		(* UPS Überwachung *)
		UPS.st_config.b_config_fertig := FALSE;
		UPS.st_config.b_station_aktiv := TRUE;
		UPS.st_config.i16_meld_startindex := 440;		(*-445*)
		UPS.st_config.str_beschreibung := ' ';
		UPS.st_config.str_instanz_name := 'UPS Überwachung';
		UPS.st_config.b_config_fertig := TRUE;

		(*Einpresskraftkontroller *)
		einpresskraft_kontroller.st_config.b_config_fertig := FALSE;
		einpresskraft_kontroller.st_config.b_station_aktiv := TRUE;
		einpresskraft_kontroller.st_config.i16_meld_startindex := 460;
		einpresskraft_kontroller.st_config.str_beschreibung := ' ';
		einpresskraft_kontroller.st_config.str_instanz_name := 'Einpresskraftkontroller';

		CASE gst_datensatz.st_md.i16_typ_zelle OF
			KEINE_ZELLE:
				gst_datensatz.st_band.st_einpressen.st_einstellungen.enu_modus := KEIN_MODUS;
			BESTUECKZELLE_1700:
				gst_datensatz.st_band.st_einpressen.st_einstellungen.enu_modus := F_MAXWERT;
			BESTUECKZELLE_1720:
				gst_datensatz.st_band.st_einpressen.st_einstellungen.enu_modus := F_MAXWERT;
			RASTERFOLIE:
				gst_datensatz.st_band.st_einpressen.st_einstellungen.enu_modus := KEIN_MODUS;
		END_CASE

		einpresskraft_kontroller.st_config.b_config_fertig := TRUE;
		
		(* Kraftmessdose Kanal 1*)
		kraftmessdose.fb.st_config.b_config_fertig := FALSE;
		kraftmessdose.fb.st_config.b_station_aktiv := TRUE;
		kraftmessdose.fb.st_config.i16_meld_startindex := 480;
		kraftmessdose.fb.st_config.str_beschreibung := ' ';
		kraftmessdose.fb.st_config.str_instanz_name := 'Kraftmessdose Kanal 1';
		kraftmessdose.fb.st_config.b_config_fertig := TRUE;
		
		(* Nockenschaltwerk Bestückachse *)
		nockenschaltwerk_bestueckachse.st_config.b_config_fertig := FALSE;
		nockenschaltwerk_bestueckachse.st_config.b_station_aktiv := TRUE;
		nockenschaltwerk_bestueckachse.st_config.i16_meld_startindex := 500;
		nockenschaltwerk_bestueckachse.st_config.str_beschreibung := ' ';
		nockenschaltwerk_bestueckachse.st_config.str_instanz_name := 'Nockenschaltwerk Bestückachse';
		nockenschaltwerk_bestueckachse.st_config.b_config_fertig := TRUE;
		
		(* Nockenschaltwerk Z-Achse *)
		(* 520 *)
		
		(* Nockenschaltwerk Y-Achse *)
		(* 540 *)
		
		(* Frei *)
		(* 560 *)

		(* Safety *)
		safety.st_config.b_config_fertig := FALSE;
		safety.st_config.b_station_aktiv := TRUE;
		safety.st_config.i16_meld_startindex := 580;
		safety.st_config.str_beschreibung := ' ';
		safety.st_config.str_instanz_name := 'Safety';
		safety.st_config.b_config_fertig := TRUE;
		
		(* XML-Server *)
		xml_server.st_config.b_config_fertig := FALSE;
		xml_server.st_config.b_station_aktiv := TRUE;
		xml_server.st_config.i16_meld_startindex := 620;
		xml_server.st_config.str_beschreibung := ' ';
		xml_server.st_config.str_instanz_name := 'XML-Server';
		xml_server.st_config.b_config_fertig := TRUE;

		(* Kurvenscheibeneditor *)
		fb_edit_mfps_bestuecken_z.st_config.b_config_fertig := FALSE;
		fb_edit_mfps_bestuecken_z.st_config.b_station_aktiv := TRUE;
		fb_edit_mfps_bestuecken_z.st_config.i16_meld_startindex := 640;
		fb_edit_mfps_bestuecken_z.st_config.str_beschreibung := ' ';
		fb_edit_mfps_bestuecken_z.st_config.str_instanz_name := 'Kurvenscheibeneditor Bestücken Z-Achse';
		fb_edit_mfps_bestuecken_z.st_config.b_config_fertig := TRUE;
		
		fb_edit_mfps_bestuecken_y.st_config.b_config_fertig := FALSE;
		fb_edit_mfps_bestuecken_y.st_config.b_station_aktiv := TRUE;
		fb_edit_mfps_bestuecken_y.st_config.i16_meld_startindex := 660;
		fb_edit_mfps_bestuecken_y.st_config.str_beschreibung := ' ';
		fb_edit_mfps_bestuecken_y.st_config.str_instanz_name := 'Kurvenscheibeneditor Bestücken Y-Achse';
		fb_edit_mfps_bestuecken_y.st_config.b_config_fertig := TRUE;
		
		fb_edit_mfps_yz_tisch.st_config.b_config_fertig := FALSE;
		fb_edit_mfps_yz_tisch.st_config.b_station_aktiv := TRUE;
		fb_edit_mfps_yz_tisch.st_config.i16_meld_startindex := 680;
		fb_edit_mfps_yz_tisch.st_config.str_beschreibung := ' ';
		fb_edit_mfps_yz_tisch.st_config.str_instanz_name := 'Kurvenscheibeneditor YZ-Tisch';
		fb_edit_mfps_yz_tisch.st_config.b_config_fertig := TRUE;

		fb_edit_mfps_bestuecken_b.st_config.b_config_fertig := FALSE;
		fb_edit_mfps_bestuecken_b.st_config.b_station_aktiv := TRUE;
		fb_edit_mfps_bestuecken_b.st_config.i16_meld_startindex := 860;
		fb_edit_mfps_bestuecken_b.st_config.str_beschreibung := ' ';
		fb_edit_mfps_bestuecken_b.st_config.str_instanz_name := 'Kurvenscheibeneditor Bestücken B-Achse';
		fb_edit_mfps_bestuecken_b.st_config.b_config_fertig := TRUE;

		fb_camtable_bestueckachse.st_config.b_config_fertig := FALSE;
		fb_camtable_bestueckachse.st_config.b_station_aktiv := TRUE;
		fb_camtable_bestueckachse.st_config.i16_meld_startindex := 880;
		fb_camtable_bestueckachse.st_config.str_beschreibung := ' ';
		fb_camtable_bestueckachse.st_config.str_instanz_name := 'Kurvenscheibeneditor Bestückachse';
		fb_camtable_bestueckachse.st_config.b_config_fertig := TRUE;

		(* Bestückbildgenerierung *)
		bbgen.st_config.b_config_fertig := FALSE;
		bbgen.st_config.b_station_aktiv := TRUE;
		bbgen.st_config.i16_meld_startindex := 700;
		bbgen.st_config.str_beschreibung := ' ';
		bbgen.st_config.str_instanz_name := 'Bestückbildgenerierung';
		bbgen.st_config.b_config_fertig := TRUE;
		
		(* Barcodereader *)
		barcode.fb.st_config.b_config_fertig := FALSE;
		barcode.fb.st_config.b_station_aktiv := TRUE;
		barcode.fb.st_config.i16_meld_startindex := 720;
		barcode.fb.st_config.str_beschreibung := ' ';
		barcode.fb.st_config.str_instanz_name := 'Barcodereader';
		barcode.fb.st_config.b_config_fertig := TRUE;
		
		(* Ballufftagreader *)
		balluff_tag_reader.fb.st_config.b_config_fertig := FALSE;
		balluff_tag_reader.fb.st_config.b_station_aktiv := TRUE;
		balluff_tag_reader.fb.st_config.i16_meld_startindex := 740;
		balluff_tag_reader.fb.st_config.str_beschreibung := ' ';
		balluff_tag_reader.fb.st_config.str_instanz_name := 'Ballufftagreader';
		balluff_tag_reader.fb.st_config.b_config_fertig := TRUE;

		(* WT-Transport Warteposition 1720 *)
		wt_transport_warteposition_1720.st_config.b_config_fertig := FALSE;
		wt_transport_warteposition_1720.st_config.i16_meld_startindex := 760;
		wt_transport_warteposition_1720.st_config.str_beschreibung := ' ';
		wt_transport_warteposition_1720.st_config.str_instanz_name := 'WT-Transport Warteposition 1720';
		wt_transport_warteposition_1720.st_config.b_config_fertig := TRUE;
		
		(* WT-Transport Beladestation 1720 *)
		wt_transport_beladen_1720.st_config.b_config_fertig := FALSE;
		wt_transport_beladen_1720.st_config.i16_meld_startindex := 780;
		wt_transport_beladen_1720.st_config.str_beschreibung := ' ';
		wt_transport_beladen_1720.st_config.str_instanz_name := 'WT-Transport Beladestation 1720';
		wt_transport_beladen_1720.st_config.b_config_fertig := TRUE;
		
		(* Rasterfolienmontge *)
		rasterfolienmontage.st_config.b_config_fertig := FALSE;
		rasterfolienmontage.st_config.b_station_aktiv := TRUE;
		rasterfolienmontage.st_config.i16_meld_startindex := 800;
		rasterfolienmontage.st_config.str_beschreibung := ' ';
		rasterfolienmontage.st_config.str_instanz_name := 'Rasterfolienmontge';
		rasterfolienmontage.st_config.b_config_fertig := TRUE;
		
		(* Rasterfolieneinzug *)
		rasterfolieneinzug.st_config.b_config_fertig := FALSE;
		rasterfolieneinzug.st_config.b_station_aktiv := TRUE;
		rasterfolieneinzug.st_config.i16_meld_startindex := 820;
		rasterfolieneinzug.st_config.str_beschreibung := ' ';
		rasterfolieneinzug.st_config.str_instanz_name := 'Rasterfolieneinzug';
		rasterfolieneinzug.st_config.b_config_fertig := TRUE;

		(*Tag lesen und schreiben *)
		Lesen_Schreiben_Tag.st_config.b_config_fertig := FALSE;
		Lesen_Schreiben_Tag.st_config.b_station_aktiv := TRUE;
		Lesen_Schreiben_Tag.st_config.i16_meld_startindex := 840;
		Lesen_Schreiben_Tag.st_config.str_beschreibung := ' ';
		Lesen_Schreiben_Tag.st_config.str_instanz_name := 'Tag lesen und schreiben';
		Lesen_Schreiben_Tag.st_config.b_config_fertig := TRUE;

		(* Wartung *)
		wartung.st_config.b_config_fertig := FALSE;
		wartung.st_config.b_station_aktiv := TRUE;
		wartung.st_config.i16_meld_startindex := 920;
		wartung.st_config.str_beschreibung := ' ';
		wartung.st_config.str_instanz_name := 'Wartung';
		wartung.st_config.b_config_fertig := TRUE;

		(*Service *)
		Service.st_config.b_config_fertig := FALSE;
		Service.st_config.b_station_aktiv := TRUE;
		Service.st_config.i16_meld_startindex := 900;
		Service.st_config.str_beschreibung := ' ';
		Service.st_config.str_instanz_name := 'Service';
		Service.st_config.b_config_fertig := TRUE;

		(*TouchProbe *)
		ST_TouchProbe.st_config.b_config_fertig := FALSE;
		ST_TouchProbe.st_config.b_station_aktiv := TRUE;
		ST_TouchProbe.st_config.i16_meld_startindex := 940;
		ST_TouchProbe.st_config.str_beschreibung := ' ';
		ST_TouchProbe.st_config.str_instanz_name := 'TouchProbe';
		ST_TouchProbe.st_config.b_config_fertig := TRUE;

		(*AutocheckinDaten *)
		ST_AutoCheckIn.fb_AutocheckinDaten.st_config.b_config_fertig:= FALSE;
		ST_AutoCheckIn.fb_AutocheckinDaten.st_config.b_station_aktiv:= TRUE;
		ST_AutoCheckIn.fb_AutocheckinDaten.st_config.i16_meld_startindex:=	960;
		ST_AutoCheckIn.fb_AutocheckinDaten.st_config.str_beschreibung:= ' ';
		ST_AutoCheckIn.fb_AutocheckinDaten.st_config.str_instanz_name:=	'AutoCheckInDaten';
		ST_AutoCheckIn.fb_AutocheckinDaten.st_config.b_config_fertig:= TRUE;

		(* WT-Transport Warteposition Achse 1700 *)
		wt_transport_warteposition_1700.st_config.b_config_fertig := FALSE;
		wt_transport_warteposition_1700.st_config.i16_meld_startindex := 400;
		wt_transport_warteposition_1700.st_config.str_beschreibung := ' ';
		wt_transport_warteposition_1700.st_config.str_instanz_name := 'WT-Transport Warteposition 1700';
		wt_transport_warteposition_1700.st_config.b_config_fertig := TRUE;
		
		(* WT-Transport Beladestation Achse 1700 *)
		wt_transport_beladen_achse_1700.st_config.b_config_fertig := FALSE;
		wt_transport_beladen_achse_1700.st_config.i16_meld_startindex := 420;
		wt_transport_beladen_achse_1700.st_config.str_beschreibung := ' ';
		wt_transport_beladen_achse_1700.st_config.str_instanz_name := 'WT-Transport Beladestation Achse 1700';
		wt_transport_beladen_achse_1700.st_config.b_config_fertig := TRUE;

		(* EtherCAT Diagnose *)
		Index:=1;
		EtherCatDiag[Index].st_config.b_config_fertig := FALSE;
		EtherCatDiag[Index].st_config.b_station_aktiv := TRUE;
		EtherCatDiag[Index].st_config.i16_meld_startindex := 980;
		EtherCatDiag[Index].st_config.str_beschreibung := ' ';
		EtherCatDiag[Index].st_config.str_instanz_name := 'Grundmaschine';
		EtherCatDiag[Index].st_config.b_config_fertig := TRUE;

		(* EtherCAT Diagnose *)
		Index:=2;
		EtherCatDiag[Index].st_config.b_config_fertig := FALSE;
		EtherCatDiag[Index].st_config.b_station_aktiv := TRUE;
		EtherCatDiag[Index].st_config.i16_meld_startindex := 985;
		EtherCatDiag[Index].st_config.str_beschreibung := ' ';
		EtherCatDiag[Index].st_config.str_instanz_name := 'Hublift links';
		EtherCatDiag[Index].st_config.b_config_fertig := TRUE;

		(* EtherCAT Diagnose *)
		Index:=3;
		EtherCatDiag[Index].st_config.b_config_fertig := FALSE;
		EtherCatDiag[Index].st_config.b_station_aktiv := TRUE;
		EtherCatDiag[Index].st_config.i16_meld_startindex := 990;
		EtherCatDiag[Index].st_config.str_beschreibung := ' ';
		EtherCatDiag[Index].st_config.str_instanz_name := 'Hublift rechts';
		EtherCatDiag[Index].st_config.b_config_fertig := TRUE;

		(* EtherCAT Diagnose *)
		Index:=4;
		EtherCatDiag[Index].st_config.b_config_fertig := FALSE;
		EtherCatDiag[Index].st_config.b_station_aktiv := TRUE;
		EtherCatDiag[Index].st_config.i16_meld_startindex := 995;
		EtherCatDiag[Index].st_config.str_beschreibung := ' ';
		EtherCatDiag[Index].st_config.str_instanz_name := 'Bandeinzug';
		EtherCatDiag[Index].st_config.b_config_fertig := TRUE;

		(* Melde-Arrays rücksetzen *)
		FOR i := 0 TO SIZEOF (garr_stoermeldungen) / SIZEOF (garr_stoermeldungen[0]) - 1 BY 1 DO
			garr_stoermeldungen[i] := 0;
		END_FOR
		FOR i := 0 TO SIZEOF (garr_betriebsmeldungen) / SIZEOF (garr_betriebsmeldungen[0]) - 1 BY 1 DO
			garr_betriebsmeldungen[i] := 0;
		END_FOR
ELSE
	b_config_fertig := TRUE;
END_IF

		
		
END_PROGRAM

(* POU Gemeinsamkeiten17xx/Initialisierung/Startup/ST_Datainit_Zylinder, ST *)
PROGRAM ST_Datainit_Zylinder
VAR
	b_config_fertig			: BOOL := FALSE;
END_VAR
IF	NOT zyl_wt_zentrierer_tisch.fb.st_config.b_config_fertig OR
	NOT zyl_wt_stopper_tisch.fb.st_config.b_config_fertig OR
	NOT zyl_wt_stopper_auslauf.fb.st_config.b_config_fertig OR
	NOT zyl_hublift_rechts_lift.fb.st_config.b_config_fertig OR
	NOT zyl_hublift_rechts_wt_einzug.fb.st_config.b_config_fertig OR
	NOT zyl_hublift_rechts_wt_klinke.fb.st_config.b_config_fertig OR
	NOT zyl_hublift_links_lift.fb.st_config.b_config_fertig OR
	NOT zyl_hublift_links_wt_einzug.fb.st_config.b_config_fertig OR
	NOT zyl_hublift_links_wt_klinke.fb.st_config.b_config_fertig OR
	NOT zyl_hublift_links_stopper.fb.st_config.b_config_fertig OR
	NOT zyl_hublift_links_eingriffschutz.fb.st_config.b_config_fertig OR
	NOT zyl_haspel_li_heben.fb.st_config.b_config_fertig OR
	NOT zyl_haspel_li_abspulen.fb.st_config.b_config_fertig OR
	NOT zyl_haspel_li_sperren.fb.st_config.b_config_fertig OR
	NOT zyl_haspel_re_heben.fb.st_config.b_config_fertig OR
	NOT zyl_haspel_re_abspulen.fb.st_config.b_config_fertig OR
	NOT zyl_haspel_re_sperren.fb.st_config.b_config_fertig OR
	NOT zyl_haspel_verschieben.fb.st_config.b_config_fertig OR
	NOT zyl_bandeinzuege_verschieben.fb.st_config.b_config_fertig OR
	NOT zyl_bawe_vorschub.fb.st_config.b_config_fertig OR
	NOT zyl_bawe_querschub.fb.st_config.b_config_fertig OR
	NOT zyl_bawe_faenger_li.fb.st_config.b_config_fertig OR
	NOT zyl_bawe_faenger_re.fb.st_config.b_config_fertig OR
	NOT zyl_bawe_halter_li.fb.st_config.b_config_fertig OR
	NOT zyl_bawe_halter_re.fb.st_config.b_config_fertig OR
	NOT zyl_wt_stopper_einlauf.fb.st_config.b_config_fertig OR
	NOT zyl_rafo_faenger.fb.st_config.b_config_fertig OR
	NOT zyl_rafo_klemmen.fb.st_config.b_config_fertig OR
	NOT zyl_rafo_vorschub.fb.st_config.b_config_fertig OR
	NOT zyl_rafo_kamm.fb.st_config.b_config_fertig OR
	NOT zyl_rafo_vorzentrierer.fb.st_config.b_config_fertig OR
	NOT zyl_Indexier_Bestueckpos.fb.st_config.b_config_fertig OR
	NOT zyl_Indexier_Einlauf.fb.st_config.b_config_fertig
	THEN

		(* WT Zentrierzylinder am Tisch *)
		zyl_wt_zentrierer_tisch.fb.st_config.b_config_fertig := FALSE;
		zyl_wt_zentrierer_tisch.fb.st_config.b_endlage1_aktiv := FALSE;
		zyl_wt_zentrierer_tisch.fb.st_config.b_endlage2_aktiv := FALSE;
		zyl_wt_zentrierer_tisch.fb.st_config.b_sensor1_aktiv := TRUE;
		zyl_wt_zentrierer_tisch.fb.st_config.b_sensor2_aktiv := TRUE;
		zyl_wt_zentrierer_tisch.fb.st_config.i16_gruppe := 3;
		zyl_wt_zentrierer_tisch.fb.st_config.i16_identnummer := 15;
		zyl_wt_zentrierer_tisch.fb.st_config.i16_meld_startindex := 2280;
		zyl_wt_zentrierer_tisch.fb.st_config.str_beschreibung := ' ';
		zyl_wt_zentrierer_tisch.fb.st_config.str_instanz_name := 'WT Zentrierzylinder am Tisch';
		zyl_wt_zentrierer_tisch.fb.st_config.str_zylinder_typ := '2V4E_EIN_AUS';
		zyl_wt_zentrierer_tisch.fb.st_config.t_ein_aus_fahrzeit := t#0ms;
		zyl_wt_zentrierer_tisch.fb.st_config.t_ueberwachungszeit := t#1000ms;
		zyl_wt_zentrierer_tisch.fb.st_config.i16_tzk_faktor_ausfahren := 100;
		zyl_wt_zentrierer_tisch.fb.st_config.i16_tzk_faktor_einfahren := 100;
		zyl_wt_zentrierer_tisch.fb.st_config.b_config_fertig := TRUE;
		
		(* WT Stoppzylinder am Tisch *)
		zyl_wt_stopper_tisch.fb.st_config.b_config_fertig := FALSE;
		zyl_wt_stopper_tisch.fb.st_config.b_endlage1_aktiv := FALSE;
		zyl_wt_stopper_tisch.fb.st_config.b_endlage2_aktiv := FALSE;
		zyl_wt_stopper_tisch.fb.st_config.b_sensor1_aktiv := TRUE;
		zyl_wt_stopper_tisch.fb.st_config.b_sensor2_aktiv := FALSE;
		zyl_wt_stopper_tisch.fb.st_config.i16_gruppe := 3;
		zyl_wt_stopper_tisch.fb.st_config.i16_identnummer := 16;
		zyl_wt_stopper_tisch.fb.st_config.i16_meld_startindex := 2300;
		zyl_wt_stopper_tisch.fb.st_config.str_beschreibung := ' ';
		zyl_wt_stopper_tisch.fb.st_config.str_instanz_name := 'WT Stoppzylinder am Tisch';

		zyl_wt_stopper_tisch.fb.st_config.t_ein_aus_fahrzeit := t#0ms;
		zyl_wt_stopper_tisch.fb.st_config.t_ueberwachungszeit := t#1000ms;
		zyl_wt_stopper_tisch.fb.st_config.i16_tzk_faktor_ausfahren := 100;
		zyl_wt_stopper_tisch.fb.st_config.i16_tzk_faktor_einfahren := 100;


		IF gst_Datensatz.st_md.b_anwahl_transport_achse THEN
			zyl_wt_stopper_tisch.fb.st_config.str_zylinder_typ := '1V0E_NO';
		ELSE
			zyl_wt_stopper_tisch.fb.st_config.str_zylinder_typ := '2V2E_EIN_AUS';
		END_IF

		zyl_wt_stopper_tisch.fb.st_config.b_config_fertig := TRUE;

		(* WT Stopperzylinder am Auslauf *)
		CASE gst_datensatz.st_md.i16_typ_zelle OF
			KEINE_ZELLE:
				;
			BESTUECKZELLE_1700, RASTERFOLIE:
				zyl_wt_stopper_auslauf.fb.st_config.b_config_fertig := FALSE;
				zyl_wt_stopper_auslauf.fb.st_config.b_endlage1_aktiv := FALSE;
				zyl_wt_stopper_auslauf.fb.st_config.b_endlage2_aktiv := FALSE;
				zyl_wt_stopper_auslauf.fb.st_config.b_sensor1_aktiv := FALSE;
				zyl_wt_stopper_auslauf.fb.st_config.b_sensor2_aktiv := FALSE;
				zyl_wt_stopper_auslauf.fb.st_config.i16_gruppe := 3;
				zyl_wt_stopper_auslauf.fb.st_config.i16_identnummer := 17;
				zyl_wt_stopper_auslauf.fb.st_config.i16_meld_startindex := 2320;
				zyl_wt_stopper_auslauf.fb.st_config.str_beschreibung := ' ';
				zyl_wt_stopper_auslauf.fb.st_config.str_instanz_name := 'WT Stopperzylinder am Auslauf';
				zyl_wt_stopper_auslauf.fb.st_config.str_zylinder_typ := '2V0E';
				zyl_wt_stopper_auslauf.fb.st_config.t_ein_aus_fahrzeit := t#150ms;
				zyl_wt_stopper_auslauf.fb.st_config.t_ueberwachungszeit := t#1000ms;
				zyl_wt_stopper_auslauf.fb.st_config.i16_tzk_faktor_ausfahren := 100;
				zyl_wt_stopper_auslauf.fb.st_config.i16_tzk_faktor_einfahren := 100;
				zyl_wt_stopper_auslauf.fb.st_config.b_config_fertig := TRUE;

			BESTUECKZELLE_1720:
				zyl_wt_stopper_auslauf.fb.st_config.b_config_fertig := FALSE;
				zyl_wt_stopper_auslauf.fb.st_config.b_endlage1_aktiv := FALSE;
				zyl_wt_stopper_auslauf.fb.st_config.b_endlage2_aktiv := FALSE;
				zyl_wt_stopper_auslauf.fb.st_config.b_sensor1_aktiv := FALSE;
				zyl_wt_stopper_auslauf.fb.st_config.b_sensor2_aktiv := FALSE;
				zyl_wt_stopper_auslauf.fb.st_config.i16_gruppe := 3;
				zyl_wt_stopper_auslauf.fb.st_config.i16_identnummer := 17;
				zyl_wt_stopper_auslauf.fb.st_config.i16_meld_startindex := 2320;
				zyl_wt_stopper_auslauf.fb.st_config.str_beschreibung := ' ';
				zyl_wt_stopper_auslauf.fb.st_config.str_instanz_name := 'WT Stopperzylinder am Auslauf';
				zyl_wt_stopper_auslauf.fb.st_config.str_zylinder_typ := '2V2E_EIN_AUS';
				zyl_wt_stopper_auslauf.fb.st_config.t_ein_aus_fahrzeit := t#150ms;
				zyl_wt_stopper_auslauf.fb.st_config.t_ueberwachungszeit := t#1000ms;
				zyl_wt_stopper_auslauf.fb.st_config.i16_tzk_faktor_ausfahren := 100;
				zyl_wt_stopper_auslauf.fb.st_config.i16_tzk_faktor_einfahren := 100;
				zyl_wt_stopper_auslauf.fb.st_config.b_config_fertig := TRUE;
		END_CASE

		(* Hublift-Lift rechts *)
		zyl_hublift_rechts_lift.fb.st_config.b_config_fertig := FALSE;
		zyl_hublift_rechts_lift.fb.st_config.b_endlage1_aktiv := TRUE;
		zyl_hublift_rechts_lift.fb.st_config.b_endlage2_aktiv := FALSE;
		zyl_hublift_rechts_lift.fb.st_config.b_sensor1_aktiv := TRUE;
		zyl_hublift_rechts_lift.fb.st_config.b_sensor2_aktiv := FALSE;
		zyl_hublift_rechts_lift.fb.st_config.i16_gruppe := 4;
		zyl_hublift_rechts_lift.fb.st_config.i16_identnummer := 18;
		zyl_hublift_rechts_lift.fb.st_config.i16_meld_startindex := 2340;
		zyl_hublift_rechts_lift.fb.st_config.str_beschreibung := ' ';
		zyl_hublift_rechts_lift.fb.st_config.str_instanz_name := 'Hublift-Lift rechts';
		zyl_hublift_rechts_lift.fb.st_config.str_zylinder_typ := '2V2E_EIN_AUS';
		zyl_hublift_rechts_lift.fb.st_config.t_ein_aus_fahrzeit := t#0ms;
		zyl_hublift_rechts_lift.fb.st_config.t_ueberwachungszeit := t#3500ms;
		zyl_hublift_rechts_lift.fb.st_config.i16_tzk_faktor_ausfahren := 100;
		zyl_hublift_rechts_lift.fb.st_config.i16_tzk_faktor_einfahren := 100;
		zyl_hublift_rechts_lift.fb.st_config.b_config_fertig := TRUE;
		
		(* Hublift-WT-Einzug rechts *)
		zyl_hublift_rechts_wt_einzug.fb.st_config.b_config_fertig := FALSE;
		zyl_hublift_rechts_wt_einzug.fb.st_config.b_endlage1_aktiv := TRUE;
		zyl_hublift_rechts_wt_einzug.fb.st_config.b_endlage2_aktiv := FALSE;
		zyl_hublift_rechts_wt_einzug.fb.st_config.b_sensor1_aktiv := TRUE;
		zyl_hublift_rechts_wt_einzug.fb.st_config.b_sensor2_aktiv := FALSE;
		zyl_hublift_rechts_wt_einzug.fb.st_config.i16_gruppe := 4;
		zyl_hublift_rechts_wt_einzug.fb.st_config.i16_identnummer := 19;
		zyl_hublift_rechts_wt_einzug.fb.st_config.i16_meld_startindex := 2360;
		zyl_hublift_rechts_wt_einzug.fb.st_config.str_beschreibung := ' ';
		zyl_hublift_rechts_wt_einzug.fb.st_config.str_instanz_name := 'Hublift-WT-Einzug rechts';
		zyl_hublift_rechts_wt_einzug.fb.st_config.str_zylinder_typ := '2V2E_EIN_AUS';
		zyl_hublift_rechts_wt_einzug.fb.st_config.t_ein_aus_fahrzeit := t#0ms;
		zyl_hublift_rechts_wt_einzug.fb.st_config.t_ueberwachungszeit := t#2500ms;
		zyl_hublift_rechts_wt_einzug.fb.st_config.i16_tzk_faktor_ausfahren := 100;
		zyl_hublift_rechts_wt_einzug.fb.st_config.i16_tzk_faktor_einfahren := 100;
		zyl_hublift_rechts_wt_einzug.fb.st_config.b_config_fertig := TRUE;
		
		(* Hublift-WT-Klinke rechts *)
		zyl_hublift_rechts_wt_klinke.fb.st_config.b_config_fertig := FALSE;
		zyl_hublift_rechts_wt_klinke.fb.st_config.b_endlage1_aktiv := TRUE;
		zyl_hublift_rechts_wt_klinke.fb.st_config.b_endlage2_aktiv := FALSE;
		zyl_hublift_rechts_wt_klinke.fb.st_config.b_sensor1_aktiv := TRUE;
		zyl_hublift_rechts_wt_klinke.fb.st_config.b_sensor2_aktiv := FALSE;
		zyl_hublift_rechts_wt_klinke.fb.st_config.i16_gruppe := 4;
		zyl_hublift_rechts_wt_klinke.fb.st_config.i16_identnummer := 20;
		zyl_hublift_rechts_wt_klinke.fb.st_config.i16_meld_startindex := 2380;
		zyl_hublift_rechts_wt_klinke.fb.st_config.str_beschreibung := ' ';
		zyl_hublift_rechts_wt_klinke.fb.st_config.str_instanz_name := 'Hublift-WT-Klinke rechts';
		zyl_hublift_rechts_wt_klinke.fb.st_config.str_zylinder_typ := '2V2E_EIN_AUS';
		zyl_hublift_rechts_wt_klinke.fb.st_config.t_ein_aus_fahrzeit := t#0ms;
		zyl_hublift_rechts_wt_klinke.fb.st_config.t_ueberwachungszeit := t#1500ms;
		zyl_hublift_rechts_wt_klinke.fb.st_config.i16_tzk_faktor_ausfahren := 100;
		zyl_hublift_rechts_wt_klinke.fb.st_config.i16_tzk_faktor_einfahren := 100;
		zyl_hublift_rechts_wt_klinke.fb.st_config.b_config_fertig := TRUE;
		
		(* Hublift-Lift links *)
		zyl_hublift_links_lift.fb.st_config.b_config_fertig := FALSE;
		zyl_hublift_links_lift.fb.st_config.b_endlage1_aktiv := TRUE;
		zyl_hublift_links_lift.fb.st_config.b_endlage2_aktiv := FALSE;
		zyl_hublift_links_lift.fb.st_config.b_sensor1_aktiv := TRUE;
		zyl_hublift_links_lift.fb.st_config.b_sensor2_aktiv := FALSE;
		zyl_hublift_links_lift.fb.st_config.i16_gruppe := 4;
		zyl_hublift_links_lift.fb.st_config.i16_identnummer := 21;
		zyl_hublift_links_lift.fb.st_config.i16_meld_startindex := 2400;
		zyl_hublift_links_lift.fb.st_config.str_beschreibung := ' ';
		zyl_hublift_links_lift.fb.st_config.str_instanz_name := 'Hublift-Lift links';
		zyl_hublift_links_lift.fb.st_config.str_zylinder_typ := '2V2E_EIN_AUS';
		zyl_hublift_links_lift.fb.st_config.t_ein_aus_fahrzeit := t#0ms;
		zyl_hublift_links_lift.fb.st_config.t_ueberwachungszeit := t#3500ms;
		zyl_hublift_links_lift.fb.st_config.i16_tzk_faktor_ausfahren := 100;
		zyl_hublift_links_lift.fb.st_config.i16_tzk_faktor_einfahren := 100;
		zyl_hublift_links_lift.fb.st_config.b_config_fertig := TRUE;
		
		(* Hublift-WT-Einzug links *)
		zyl_hublift_links_wt_einzug.fb.st_config.b_config_fertig := FALSE;
		zyl_hublift_links_wt_einzug.fb.st_config.b_endlage1_aktiv := TRUE;
		zyl_hublift_links_wt_einzug.fb.st_config.b_endlage2_aktiv := FALSE;
		zyl_hublift_links_wt_einzug.fb.st_config.b_sensor1_aktiv := TRUE;
		zyl_hublift_links_wt_einzug.fb.st_config.b_sensor2_aktiv := FALSE;
		zyl_hublift_links_wt_einzug.fb.st_config.i16_gruppe := 4;
		zyl_hublift_links_wt_einzug.fb.st_config.i16_identnummer := 22;
		zyl_hublift_links_wt_einzug.fb.st_config.i16_meld_startindex := 2420;
		zyl_hublift_links_wt_einzug.fb.st_config.str_beschreibung := ' ';
		zyl_hublift_links_wt_einzug.fb.st_config.str_instanz_name := 'Hublift-WT-Einzug links';
		zyl_hublift_links_wt_einzug.fb.st_config.str_zylinder_typ := '2V2E_EIN_AUS';
		zyl_hublift_links_wt_einzug.fb.st_config.t_ein_aus_fahrzeit := t#0ms;
		zyl_hublift_links_wt_einzug.fb.st_config.t_ueberwachungszeit := t#2500ms;
		zyl_hublift_links_wt_einzug.fb.st_config.i16_tzk_faktor_ausfahren := 100;
		zyl_hublift_links_wt_einzug.fb.st_config.i16_tzk_faktor_einfahren := 100;
		zyl_hublift_links_wt_einzug.fb.st_config.b_config_fertig := TRUE;

		(* Hublift-WT-Klinke links *)
		zyl_hublift_links_wt_klinke.fb.st_config.b_config_fertig := FALSE;
		zyl_hublift_links_wt_klinke.fb.st_config.b_endlage1_aktiv := TRUE;
		zyl_hublift_links_wt_klinke.fb.st_config.b_endlage2_aktiv := FALSE;
		zyl_hublift_links_wt_klinke.fb.st_config.b_sensor1_aktiv := TRUE;
		zyl_hublift_links_wt_klinke.fb.st_config.b_sensor2_aktiv := FALSE;
		zyl_hublift_links_wt_klinke.fb.st_config.i16_gruppe := 4;
		zyl_hublift_links_wt_klinke.fb.st_config.i16_identnummer := 23;
		zyl_hublift_links_wt_klinke.fb.st_config.i16_meld_startindex := 2440;
		zyl_hublift_links_wt_klinke.fb.st_config.str_beschreibung := ' ';
		zyl_hublift_links_wt_klinke.fb.st_config.str_instanz_name := 'Hublift-WT-Klinke links';
		zyl_hublift_links_wt_klinke.fb.st_config.str_zylinder_typ := '2V2E_EIN_AUS';
		zyl_hublift_links_wt_klinke.fb.st_config.t_ein_aus_fahrzeit := t#0ms;
		zyl_hublift_links_wt_klinke.fb.st_config.t_ueberwachungszeit := t#1500ms;
		zyl_hublift_links_wt_klinke.fb.st_config.i16_tzk_faktor_ausfahren := 100;
		zyl_hublift_links_wt_klinke.fb.st_config.i16_tzk_faktor_einfahren := 100;
		zyl_hublift_links_wt_klinke.fb.st_config.b_config_fertig := TRUE;

		(* Hublift-Stopper links *)
		zyl_hublift_links_stopper.fb.st_config.b_config_fertig := FALSE;
		zyl_hublift_links_stopper.fb.st_config.b_endlage1_aktiv := TRUE;
		zyl_hublift_links_stopper.fb.st_config.b_endlage2_aktiv := FALSE;
		zyl_hublift_links_stopper.fb.st_config.b_sensor1_aktiv := TRUE;
		zyl_hublift_links_stopper.fb.st_config.b_sensor2_aktiv := FALSE;
		zyl_hublift_links_stopper.fb.st_config.i16_gruppe := 4;
		zyl_hublift_links_stopper.fb.st_config.i16_identnummer := 24;
		zyl_hublift_links_stopper.fb.st_config.i16_meld_startindex := 2460;
		zyl_hublift_links_stopper.fb.st_config.str_beschreibung := ' ';
		zyl_hublift_links_stopper.fb.st_config.str_instanz_name := 'Hublift-Stopper links';
		zyl_hublift_links_stopper.fb.st_config.str_zylinder_typ := '2V2E_EIN_AUS';
		zyl_hublift_links_stopper.fb.st_config.t_ein_aus_fahrzeit := t#0ms;
		zyl_hublift_links_stopper.fb.st_config.t_ueberwachungszeit := t#2000ms;
		zyl_hublift_links_stopper.fb.st_config.i16_tzk_faktor_ausfahren := 100;
		zyl_hublift_links_stopper.fb.st_config.i16_tzk_faktor_einfahren := 100;
		zyl_hublift_links_stopper.fb.st_config.b_config_fertig := TRUE;

		(* zyl_hublift_links_eingriffschutz *)
		zyl_hublift_links_eingriffschutz.fb.st_config.b_config_fertig := FALSE;
		zyl_hublift_links_eingriffschutz.fb.st_config.b_endlage1_aktiv := TRUE;
		zyl_hublift_links_eingriffschutz.fb.st_config.b_endlage2_aktiv := FALSE;
		zyl_hublift_links_eingriffschutz.fb.st_config.b_sensor1_aktiv := TRUE;
		zyl_hublift_links_eingriffschutz.fb.st_config.b_sensor2_aktiv := FALSE;
		zyl_hublift_links_eingriffschutz.fb.st_config.i16_gruppe := 4;
		zyl_hublift_links_eingriffschutz.fb.st_config.i16_identnummer := 44;
		zyl_hublift_links_eingriffschutz.fb.st_config.i16_meld_startindex := 2860;
		zyl_hublift_links_eingriffschutz.fb.st_config.str_beschreibung := ' ';
		zyl_hublift_links_eingriffschutz.fb.st_config.str_instanz_name := 'Hublift links Eingriffschutz';
		zyl_hublift_links_eingriffschutz.fb.st_config.str_zylinder_typ := '2V2E_EIN_AUS';
		zyl_hublift_links_eingriffschutz.fb.st_config.t_ein_aus_fahrzeit := t#0ms;
		zyl_hublift_links_eingriffschutz.fb.st_config.t_ueberwachungszeit := t#4000ms;
		zyl_hublift_links_eingriffschutz.fb.st_config.i16_tzk_faktor_ausfahren := 100;
		zyl_hublift_links_eingriffschutz.fb.st_config.i16_tzk_faktor_einfahren := 100;
		zyl_hublift_links_eingriffschutz.fb.st_config.b_config_fertig := TRUE;
		
		(* Haspel links heben *)
		zyl_haspel_li_heben.fb.st_config.b_config_fertig := FALSE;
		zyl_haspel_li_heben.fb.st_config.b_endlage1_aktiv := FALSE;
		zyl_haspel_li_heben.fb.st_config.b_endlage2_aktiv := FALSE;
		zyl_haspel_li_heben.fb.st_config.b_sensor1_aktiv := FALSE;
		zyl_haspel_li_heben.fb.st_config.b_sensor2_aktiv := FALSE;
		zyl_haspel_li_heben.fb.st_config.i16_gruppe := 2;
		zyl_haspel_li_heben.fb.st_config.i16_identnummer := 7;
		zyl_haspel_li_heben.fb.st_config.i16_meld_startindex := 2120;
		zyl_haspel_li_heben.fb.st_config.str_beschreibung := ' ';
		zyl_haspel_li_heben.fb.st_config.str_instanz_name := 'Haspel links heben';
		zyl_haspel_li_heben.fb.st_config.str_zylinder_typ := '2V1E_AUS';
		zyl_haspel_li_heben.fb.st_config.t_ein_aus_fahrzeit := t#0ms;
		zyl_haspel_li_heben.fb.st_config.t_ueberwachungszeit := t#8s;
		zyl_haspel_li_heben.fb.st_config.i16_tzk_faktor_ausfahren := 100;
		zyl_haspel_li_heben.fb.st_config.i16_tzk_faktor_einfahren := 100;
		zyl_haspel_li_heben.fb.st_config.b_config_fertig := TRUE;
		
		(* Haspel links abspulen *)
		zyl_haspel_li_abspulen.fb.st_config.b_config_fertig := FALSE;
		zyl_haspel_li_abspulen.fb.st_config.b_endlage1_aktiv := FALSE;
		zyl_haspel_li_abspulen.fb.st_config.b_endlage2_aktiv := FALSE;
		zyl_haspel_li_abspulen.fb.st_config.b_sensor1_aktiv := FALSE;
		zyl_haspel_li_abspulen.fb.st_config.b_sensor2_aktiv := FALSE;
		zyl_haspel_li_abspulen.fb.st_config.i16_gruppe := 2;
		zyl_haspel_li_abspulen.fb.st_config.i16_identnummer := 8;
		zyl_haspel_li_abspulen.fb.st_config.i16_meld_startindex := 2140;
		zyl_haspel_li_abspulen.fb.st_config.str_beschreibung := ' ';
		zyl_haspel_li_abspulen.fb.st_config.str_instanz_name := 'Haspel links abspulen';
		zyl_haspel_li_abspulen.fb.st_config.str_zylinder_typ := '2V1E_AUS';
		zyl_haspel_li_abspulen.fb.st_config.t_ein_aus_fahrzeit := t#0ms;
		zyl_haspel_li_abspulen.fb.st_config.t_ueberwachungszeit := t#3s;
		zyl_haspel_li_abspulen.fb.st_config.i16_tzk_faktor_ausfahren := 100;
		zyl_haspel_li_abspulen.fb.st_config.i16_tzk_faktor_einfahren := 100;
		zyl_haspel_li_abspulen.fb.st_config.b_config_fertig := TRUE;
		
		(* Haspel links sperren *)
		zyl_haspel_li_sperren.fb.st_config.b_config_fertig := FALSE;
		zyl_haspel_li_sperren.fb.st_config.b_endlage1_aktiv := FALSE;
		zyl_haspel_li_sperren.fb.st_config.b_endlage2_aktiv := FALSE;
		zyl_haspel_li_sperren.fb.st_config.b_sensor1_aktiv := TRUE;
		zyl_haspel_li_sperren.fb.st_config.b_sensor2_aktiv := FALSE;
		zyl_haspel_li_sperren.fb.st_config.i16_gruppe := 2;
		zyl_haspel_li_sperren.fb.st_config.i16_identnummer := 9;
		zyl_haspel_li_sperren.fb.st_config.i16_meld_startindex := 2160;
		zyl_haspel_li_sperren.fb.st_config.str_beschreibung := ' ';
		zyl_haspel_li_sperren.fb.st_config.str_instanz_name := 'Haspel links sperren';
		zyl_haspel_li_sperren.fb.st_config.str_zylinder_typ := '2V2E_EIN_AUS';
		zyl_haspel_li_sperren.fb.st_config.t_ein_aus_fahrzeit := t#0ms;
		zyl_haspel_li_sperren.fb.st_config.t_ueberwachungszeit := t#1000ms;
		zyl_haspel_li_sperren.fb.st_config.i16_tzk_faktor_ausfahren := 100;
		zyl_haspel_li_sperren.fb.st_config.i16_tzk_faktor_einfahren := 100;
		zyl_haspel_li_sperren.fb.st_config.b_config_fertig := TRUE;
		
		(* Haspel rechts heben *)
		zyl_haspel_re_heben.fb.st_config.b_config_fertig := FALSE;
		zyl_haspel_re_heben.fb.st_config.b_endlage1_aktiv := FALSE;
		zyl_haspel_re_heben.fb.st_config.b_endlage2_aktiv := FALSE;
		zyl_haspel_re_heben.fb.st_config.b_sensor1_aktiv := FALSE;
		zyl_haspel_re_heben.fb.st_config.b_sensor2_aktiv := FALSE;
		zyl_haspel_re_heben.fb.st_config.i16_gruppe := 2;
		zyl_haspel_re_heben.fb.st_config.i16_identnummer := 10;
		zyl_haspel_re_heben.fb.st_config.i16_meld_startindex := 2180;
		zyl_haspel_re_heben.fb.st_config.str_beschreibung := ' ';
		zyl_haspel_re_heben.fb.st_config.str_instanz_name := 'Haspel rechts heben';
		zyl_haspel_re_heben.fb.st_config.str_zylinder_typ := '2V1E_AUS';
		zyl_haspel_re_heben.fb.st_config.t_ein_aus_fahrzeit := t#0ms;
		zyl_haspel_re_heben.fb.st_config.t_ueberwachungszeit := t#8s;
		zyl_haspel_re_heben.fb.st_config.i16_tzk_faktor_ausfahren := 100;
		zyl_haspel_re_heben.fb.st_config.i16_tzk_faktor_einfahren := 100;
		zyl_haspel_re_heben.fb.st_config.b_config_fertig := TRUE;
		
		(* Haspel rechts abspulen *)
		zyl_haspel_re_abspulen.fb.st_config.b_config_fertig := FALSE;
		zyl_haspel_re_abspulen.fb.st_config.b_endlage1_aktiv := FALSE;
		zyl_haspel_re_abspulen.fb.st_config.b_endlage2_aktiv := FALSE;
		zyl_haspel_re_abspulen.fb.st_config.b_sensor1_aktiv := FALSE;
		zyl_haspel_re_abspulen.fb.st_config.b_sensor2_aktiv := FALSE;
		zyl_haspel_re_abspulen.fb.st_config.i16_gruppe := 2;
		zyl_haspel_re_abspulen.fb.st_config.i16_identnummer := 11;
		zyl_haspel_re_abspulen.fb.st_config.i16_meld_startindex := 2200;
		zyl_haspel_re_abspulen.fb.st_config.str_beschreibung := ' ';
		zyl_haspel_re_abspulen.fb.st_config.str_instanz_name := 'Haspel rechts abspulen';
		zyl_haspel_re_abspulen.fb.st_config.str_zylinder_typ := '2V1E_AUS';
		zyl_haspel_re_abspulen.fb.st_config.t_ein_aus_fahrzeit := t#0ms;
		zyl_haspel_re_abspulen.fb.st_config.t_ueberwachungszeit := t#3s;
		zyl_haspel_re_abspulen.fb.st_config.i16_tzk_faktor_ausfahren := 100;
		zyl_haspel_re_abspulen.fb.st_config.i16_tzk_faktor_einfahren := 100;
		zyl_haspel_re_abspulen.fb.st_config.b_config_fertig := TRUE;
		
		(* Haspel rechts sperren *)
		zyl_haspel_re_sperren.fb.st_config.b_config_fertig := FALSE;
		zyl_haspel_re_sperren.fb.st_config.b_endlage1_aktiv := FALSE;
		zyl_haspel_re_sperren.fb.st_config.b_endlage2_aktiv := FALSE;
		zyl_haspel_re_sperren.fb.st_config.b_sensor1_aktiv := FALSE;
		zyl_haspel_re_sperren.fb.st_config.b_sensor2_aktiv := FALSE;
		zyl_haspel_re_sperren.fb.st_config.i16_gruppe := 2;
		zyl_haspel_re_sperren.fb.st_config.i16_identnummer := 12;
		zyl_haspel_re_sperren.fb.st_config.i16_meld_startindex := 2220;
		zyl_haspel_re_sperren.fb.st_config.str_beschreibung := ' ';
		zyl_haspel_re_sperren.fb.st_config.str_instanz_name := 'Haspel rechts sperren';
		zyl_haspel_re_sperren.fb.st_config.str_zylinder_typ := '2V2E_EIN_AUS';
		zyl_haspel_re_sperren.fb.st_config.t_ein_aus_fahrzeit := t#0ms;
		zyl_haspel_re_sperren.fb.st_config.t_ueberwachungszeit := t#1000ms;
		zyl_haspel_re_sperren.fb.st_config.i16_tzk_faktor_ausfahren := 100;
		zyl_haspel_re_sperren.fb.st_config.i16_tzk_faktor_einfahren := 100;
		zyl_haspel_re_sperren.fb.st_config.b_config_fertig := TRUE;
		
		(* Haspel verschieben *)
		zyl_haspel_verschieben.fb.st_config.b_config_fertig := FALSE;
		zyl_haspel_verschieben.fb.st_config.b_endlage1_aktiv := FALSE;
		zyl_haspel_verschieben.fb.st_config.b_endlage2_aktiv := FALSE;
		zyl_haspel_verschieben.fb.st_config.b_sensor1_aktiv := TRUE;
		zyl_haspel_verschieben.fb.st_config.b_sensor2_aktiv := FALSE;
		zyl_haspel_verschieben.fb.st_config.i16_gruppe := 2;
		zyl_haspel_verschieben.fb.st_config.i16_identnummer := 13;
		zyl_haspel_verschieben.fb.st_config.i16_meld_startindex := 2240;
		zyl_haspel_verschieben.fb.st_config.str_beschreibung := ' ';
		zyl_haspel_verschieben.fb.st_config.str_instanz_name := 'Haspel verschieben';
		zyl_haspel_verschieben.fb.st_config.str_zylinder_typ := '2V2E_EIN_AUS';
		zyl_haspel_verschieben.fb.st_config.t_ein_aus_fahrzeit := t#0ms;
		zyl_haspel_verschieben.fb.st_config.t_ueberwachungszeit := t#8s;
		zyl_haspel_verschieben.fb.st_config.i16_tzk_faktor_ausfahren := 100;
		zyl_haspel_verschieben.fb.st_config.i16_tzk_faktor_einfahren := 100;
		zyl_haspel_verschieben.fb.st_config.b_config_fertig := TRUE;
		
		(* Bandeinzüge verschieben *)
		zyl_bandeinzuege_verschieben.fb.st_config.b_config_fertig := FALSE;
		zyl_bandeinzuege_verschieben.fb.st_config.b_endlage1_aktiv := FALSE;
		zyl_bandeinzuege_verschieben.fb.st_config.b_endlage2_aktiv := FALSE;
		zyl_bandeinzuege_verschieben.fb.st_config.b_sensor1_aktiv := TRUE;
		zyl_bandeinzuege_verschieben.fb.st_config.b_sensor2_aktiv := FALSE;
		zyl_bandeinzuege_verschieben.fb.st_config.i16_gruppe := 2;
		zyl_bandeinzuege_verschieben.fb.st_config.i16_identnummer := 14;
		zyl_bandeinzuege_verschieben.fb.st_config.i16_meld_startindex := 2260;
		zyl_bandeinzuege_verschieben.fb.st_config.str_beschreibung := ' ';
		zyl_bandeinzuege_verschieben.fb.st_config.str_instanz_name := 'Bandeinzüge verschieben';
		zyl_bandeinzuege_verschieben.fb.st_config.str_zylinder_typ := '2V2E_EIN_AUS';
		zyl_bandeinzuege_verschieben.fb.st_config.t_ein_aus_fahrzeit := t#0ms;
		zyl_bandeinzuege_verschieben.fb.st_config.t_ueberwachungszeit := t#8000ms;
		zyl_bandeinzuege_verschieben.fb.st_config.i16_tzk_faktor_ausfahren := 100;
		zyl_bandeinzuege_verschieben.fb.st_config.i16_tzk_faktor_einfahren := 100;
		zyl_bandeinzuege_verschieben.fb.st_config.b_config_fertig := TRUE;
		
		(* Bandwechselvorschub *)
		zyl_bawe_vorschub.fb.st_config.b_config_fertig := FALSE;
		zyl_bawe_vorschub.fb.st_config.b_endlage1_aktiv := FALSE;
		zyl_bawe_vorschub.fb.st_config.b_endlage2_aktiv := FALSE;
		zyl_bawe_vorschub.fb.st_config.b_sensor1_aktiv := FALSE;
		zyl_bawe_vorschub.fb.st_config.b_sensor2_aktiv := FALSE;
		zyl_bawe_vorschub.fb.st_config.i16_gruppe := 5;
		zyl_bawe_vorschub.fb.st_config.i16_identnummer := 25;
		zyl_bawe_vorschub.fb.st_config.i16_meld_startindex := 2480;
		zyl_bawe_vorschub.fb.st_config.str_beschreibung := ' ';
		zyl_bawe_vorschub.fb.st_config.str_instanz_name := 'Bandwechselvorschub';
		zyl_bawe_vorschub.fb.st_config.str_zylinder_typ := '2V2E_EIN_AUS';
		zyl_bawe_vorschub.fb.st_config.t_ein_aus_fahrzeit := t#0ms;
		zyl_bawe_vorschub.fb.st_config.t_ueberwachungszeit := t#2000ms;
		zyl_bawe_vorschub.fb.st_config.i16_tzk_faktor_ausfahren := 100;
		zyl_bawe_vorschub.fb.st_config.i16_tzk_faktor_einfahren := 100;
		zyl_bawe_vorschub.fb.st_config.b_config_fertig := TRUE;
		
		(* Bandwechselquerschub *)
		zyl_bawe_querschub.fb.st_config.b_config_fertig := FALSE;
		zyl_bawe_querschub.fb.st_config.b_endlage1_aktiv := FALSE;
		zyl_bawe_querschub.fb.st_config.b_endlage2_aktiv := FALSE;
		zyl_bawe_querschub.fb.st_config.b_sensor1_aktiv := FALSE;
		zyl_bawe_querschub.fb.st_config.b_sensor2_aktiv := FALSE;
		zyl_bawe_querschub.fb.st_config.i16_gruppe := 5;
		zyl_bawe_querschub.fb.st_config.i16_identnummer := 26;
		zyl_bawe_querschub.fb.st_config.i16_meld_startindex := 2500;
		zyl_bawe_querschub.fb.st_config.str_beschreibung := ' ';
		zyl_bawe_querschub.fb.st_config.str_instanz_name := 'Bandwechselquerschub';
		zyl_bawe_querschub.fb.st_config.str_zylinder_typ := '2V2E_EIN_AUS';
		zyl_bawe_querschub.fb.st_config.t_ein_aus_fahrzeit := t#0ms;
		zyl_bawe_querschub.fb.st_config.t_ueberwachungszeit := t#8000ms;
		zyl_bawe_querschub.fb.st_config.i16_tzk_faktor_ausfahren := 100;
		zyl_bawe_querschub.fb.st_config.i16_tzk_faktor_einfahren := 100;
		zyl_bawe_querschub.fb.st_config.b_config_fertig := TRUE;
		
		(* Bandwechselfänger links *)
		zyl_bawe_faenger_li.fb.st_config.b_config_fertig := FALSE;
		zyl_bawe_faenger_li.fb.st_config.b_endlage1_aktiv := FALSE;
		zyl_bawe_faenger_li.fb.st_config.b_endlage2_aktiv := FALSE;
		zyl_bawe_faenger_li.fb.st_config.b_sensor1_aktiv := FALSE;
		zyl_bawe_faenger_li.fb.st_config.b_sensor2_aktiv := FALSE;
		zyl_bawe_faenger_li.fb.st_config.i16_gruppe := 5;
		zyl_bawe_faenger_li.fb.st_config.i16_identnummer := 27;
		zyl_bawe_faenger_li.fb.st_config.i16_meld_startindex := 2520;
		zyl_bawe_faenger_li.fb.st_config.str_beschreibung := ' ';
		zyl_bawe_faenger_li.fb.st_config.str_instanz_name := 'Bandwechselfaenger links';
		zyl_bawe_faenger_li.fb.st_config.str_zylinder_typ := '2V0E';
		zyl_bawe_faenger_li.fb.st_config.t_ein_aus_fahrzeit := t#200ms;
		zyl_bawe_faenger_li.fb.st_config.t_ueberwachungszeit := t#500ms;
		zyl_bawe_faenger_li.fb.st_config.i16_tzk_faktor_ausfahren := 100;
		zyl_bawe_faenger_li.fb.st_config.i16_tzk_faktor_einfahren := 100;
		zyl_bawe_faenger_li.fb.st_config.b_config_fertig := TRUE;
		
		(* Bandwechselfänger rechts *)
		zyl_bawe_faenger_re.fb.st_config.b_config_fertig := FALSE;
		zyl_bawe_faenger_re.fb.st_config.b_endlage1_aktiv := FALSE;
		zyl_bawe_faenger_re.fb.st_config.b_endlage2_aktiv := FALSE;
		zyl_bawe_faenger_re.fb.st_config.b_sensor1_aktiv := FALSE;
		zyl_bawe_faenger_re.fb.st_config.b_sensor2_aktiv := FALSE;
		zyl_bawe_faenger_re.fb.st_config.i16_gruppe := 5;
		zyl_bawe_faenger_re.fb.st_config.i16_identnummer := 28;
		zyl_bawe_faenger_re.fb.st_config.i16_meld_startindex := 2540;
		zyl_bawe_faenger_re.fb.st_config.str_beschreibung := ' ';
		zyl_bawe_faenger_re.fb.st_config.str_instanz_name := 'Bandwechselfaenger rechts';
		zyl_bawe_faenger_re.fb.st_config.str_zylinder_typ := '2V0E';
		zyl_bawe_faenger_re.fb.st_config.t_ein_aus_fahrzeit := t#200ms;
		zyl_bawe_faenger_re.fb.st_config.t_ueberwachungszeit := t#500ms;
		zyl_bawe_faenger_re.fb.st_config.i16_tzk_faktor_ausfahren := 100;
		zyl_bawe_faenger_re.fb.st_config.i16_tzk_faktor_einfahren := 100;
		zyl_bawe_faenger_re.fb.st_config.b_config_fertig := TRUE;
		
		(* Bandwechselhalter links *)
		zyl_bawe_halter_li.fb.st_config.b_config_fertig := FALSE;
		zyl_bawe_halter_li.fb.st_config.b_endlage1_aktiv := FALSE;
		zyl_bawe_halter_li.fb.st_config.b_endlage2_aktiv := FALSE;
		zyl_bawe_halter_li.fb.st_config.b_sensor1_aktiv := FALSE;
		zyl_bawe_halter_li.fb.st_config.b_sensor2_aktiv := FALSE;
		zyl_bawe_halter_li.fb.st_config.i16_gruppe := 5;
		zyl_bawe_halter_li.fb.st_config.i16_identnummer := 29;
		zyl_bawe_halter_li.fb.st_config.i16_meld_startindex := 2560;
		zyl_bawe_halter_li.fb.st_config.str_beschreibung := ' ';
		zyl_bawe_halter_li.fb.st_config.str_instanz_name := 'Bandwechselhalter links';
		zyl_bawe_halter_li.fb.st_config.str_zylinder_typ := '2V0E';
		zyl_bawe_halter_li.fb.st_config.t_ein_aus_fahrzeit := t#200ms;
		zyl_bawe_halter_li.fb.st_config.t_ueberwachungszeit := t#500ms;
		zyl_bawe_halter_li.fb.st_config.i16_tzk_faktor_ausfahren := 100;
		zyl_bawe_halter_li.fb.st_config.i16_tzk_faktor_einfahren := 100;
		zyl_bawe_halter_li.fb.st_config.b_config_fertig := TRUE;
		
		(* Bandwechselhalter rechts *)
		zyl_bawe_halter_re.fb.st_config.b_config_fertig := FALSE;
		zyl_bawe_halter_re.fb.st_config.b_endlage1_aktiv := FALSE;
		zyl_bawe_halter_re.fb.st_config.b_endlage2_aktiv := FALSE;
		zyl_bawe_halter_re.fb.st_config.b_sensor1_aktiv := FALSE;
		zyl_bawe_halter_re.fb.st_config.b_sensor2_aktiv := FALSE;
		zyl_bawe_halter_re.fb.st_config.i16_gruppe := 5;
		zyl_bawe_halter_re.fb.st_config.i16_identnummer := 30;
		zyl_bawe_halter_re.fb.st_config.i16_meld_startindex := 2580;
		zyl_bawe_halter_re.fb.st_config.str_beschreibung := ' ';
		zyl_bawe_halter_re.fb.st_config.str_instanz_name := 'Bandwechselhalter rechts';
		zyl_bawe_halter_re.fb.st_config.str_zylinder_typ := '2V0E';
		zyl_bawe_halter_re.fb.st_config.t_ein_aus_fahrzeit := t#200ms;
		zyl_bawe_halter_re.fb.st_config.t_ueberwachungszeit := t#500ms;
		zyl_bawe_halter_re.fb.st_config.i16_tzk_faktor_ausfahren := 100;
		zyl_bawe_halter_re.fb.st_config.i16_tzk_faktor_einfahren := 100;
		zyl_bawe_halter_re.fb.st_config.b_config_fertig := TRUE;

		(* WT Stopperzylinder am Einlauf *)
		zyl_wt_stopper_einlauf.fb.st_config.b_config_fertig := FALSE;
		zyl_wt_stopper_einlauf.fb.st_config.b_endlage1_aktiv := FALSE;
		zyl_wt_stopper_einlauf.fb.st_config.b_endlage2_aktiv := FALSE;
		zyl_wt_stopper_einlauf.fb.st_config.b_sensor1_aktiv := TRUE;
		zyl_wt_stopper_einlauf.fb.st_config.b_sensor2_aktiv := TRUE;
		zyl_wt_stopper_einlauf.fb.st_config.i16_gruppe := 3;
		zyl_wt_stopper_einlauf.fb.st_config.i16_identnummer := 36;
		zyl_wt_stopper_einlauf.fb.st_config.i16_meld_startindex := 2700;
		zyl_wt_stopper_einlauf.fb.st_config.str_beschreibung := ' ';
		zyl_wt_stopper_einlauf.fb.st_config.str_instanz_name := 'WT Stopperzylinder am Einlauf';
		zyl_wt_stopper_einlauf.fb.st_config.str_zylinder_typ := '1V2E_EIN_AUS';
		zyl_wt_stopper_einlauf.fb.st_config.t_ein_aus_fahrzeit := t#0ms;
		zyl_wt_stopper_einlauf.fb.st_config.t_ueberwachungszeit := t#1000ms;
		zyl_wt_stopper_einlauf.fb.st_config.i16_tzk_faktor_ausfahren := 100;
		zyl_wt_stopper_einlauf.fb.st_config.i16_tzk_faktor_einfahren := 100;
		zyl_wt_stopper_einlauf.fb.st_config.b_config_fertig := TRUE;

		(* Rasterfolien Fänger *)
		zyl_rafo_faenger.fb.st_config.b_config_fertig := FALSE;
		zyl_rafo_faenger.fb.st_config.b_endlage1_aktiv := TRUE;
		zyl_rafo_faenger.fb.st_config.b_endlage2_aktiv := FALSE;
		zyl_rafo_faenger.fb.st_config.b_sensor1_aktiv := TRUE;
		zyl_rafo_faenger.fb.st_config.b_sensor2_aktiv := FALSE;
		zyl_rafo_faenger.fb.st_config.i16_gruppe := 7;
		zyl_rafo_faenger.fb.st_config.i16_identnummer := 37;
		zyl_rafo_faenger.fb.st_config.i16_meld_startindex := 2720;
		zyl_rafo_faenger.fb.st_config.str_beschreibung := ' ';
		zyl_rafo_faenger.fb.st_config.str_instanz_name := 'Rasterfolien Fänger';
		zyl_rafo_faenger.fb.st_config.str_zylinder_typ := '2V1E_AUS';
		zyl_rafo_faenger.fb.st_config.t_ein_aus_fahrzeit := t#100ms;
		zyl_rafo_faenger.fb.st_config.t_ueberwachungszeit := t#500ms;
		zyl_rafo_faenger.fb.st_config.i16_tzk_faktor_ausfahren := 100;
		zyl_rafo_faenger.fb.st_config.i16_tzk_faktor_einfahren := 100;
		zyl_rafo_faenger.fb.st_config.b_config_fertig := TRUE;
		
		(* Rasterfolie Klemmen *)
		zyl_rafo_klemmen.fb.st_config.b_config_fertig := FALSE;
		zyl_rafo_klemmen.fb.st_config.b_endlage1_aktiv := TRUE;
		zyl_rafo_klemmen.fb.st_config.b_endlage2_aktiv := FALSE;
		zyl_rafo_klemmen.fb.st_config.b_sensor1_aktiv := TRUE;
		zyl_rafo_klemmen.fb.st_config.b_sensor2_aktiv := FALSE;
		zyl_rafo_klemmen.fb.st_config.i16_gruppe := 7;
		zyl_rafo_klemmen.fb.st_config.i16_identnummer := 38;
		zyl_rafo_klemmen.fb.st_config.i16_meld_startindex := 2740;
		zyl_rafo_klemmen.fb.st_config.str_beschreibung := ' ';
		zyl_rafo_klemmen.fb.st_config.str_instanz_name := 'Rasterfolie Klemmen';
		zyl_rafo_klemmen.fb.st_config.str_zylinder_typ := '2V1E_AUS';
		zyl_rafo_klemmen.fb.st_config.t_ein_aus_fahrzeit := t#100ms;
		zyl_rafo_klemmen.fb.st_config.t_ueberwachungszeit := t#500ms;
		zyl_rafo_klemmen.fb.st_config.i16_tzk_faktor_ausfahren := 100;
		zyl_rafo_klemmen.fb.st_config.i16_tzk_faktor_einfahren := 100;
		zyl_rafo_klemmen.fb.st_config.b_config_fertig := TRUE;
		
		(* Rasterfolien Vorschub *)
		zyl_rafo_vorschub.fb.st_config.b_config_fertig := FALSE;
		zyl_rafo_vorschub.fb.st_config.b_endlage1_aktiv := TRUE;
		zyl_rafo_vorschub.fb.st_config.b_endlage2_aktiv := FALSE;
		zyl_rafo_vorschub.fb.st_config.b_sensor1_aktiv := TRUE;
		zyl_rafo_vorschub.fb.st_config.b_sensor2_aktiv := FALSE;
		zyl_rafo_vorschub.fb.st_config.i16_gruppe := 7;
		zyl_rafo_vorschub.fb.st_config.i16_identnummer := 39;
		zyl_rafo_vorschub.fb.st_config.i16_meld_startindex := 2760;
		zyl_rafo_vorschub.fb.st_config.str_beschreibung := ' ';
		zyl_rafo_vorschub.fb.st_config.str_instanz_name := 'Rasterplatte Wenden';
		zyl_rafo_vorschub.fb.st_config.str_zylinder_typ := '2V2E_EIN_AUS';
		zyl_rafo_vorschub.fb.st_config.t_ein_aus_fahrzeit := t#100ms;
		zyl_rafo_vorschub.fb.st_config.t_ueberwachungszeit := t#2000ms;
		zyl_rafo_vorschub.fb.st_config.i16_tzk_faktor_ausfahren := 100;
		zyl_rafo_vorschub.fb.st_config.i16_tzk_faktor_einfahren := 100;
		zyl_rafo_vorschub.fb.st_config.b_config_fertig := TRUE;
		
		(* Rasterfolien Kamm *)
		zyl_rafo_kamm.fb.st_config.b_config_fertig := FALSE;
		zyl_rafo_kamm.fb.st_config.b_endlage1_aktiv := TRUE;
		zyl_rafo_kamm.fb.st_config.b_endlage2_aktiv := FALSE;
		zyl_rafo_kamm.fb.st_config.b_sensor1_aktiv := TRUE;
		zyl_rafo_kamm.fb.st_config.b_sensor2_aktiv := FALSE;
		zyl_rafo_kamm.fb.st_config.i16_gruppe := 7;
		zyl_rafo_kamm.fb.st_config.i16_identnummer := 40;
		zyl_rafo_kamm.fb.st_config.i16_meld_startindex := 2780;
		zyl_rafo_kamm.fb.st_config.str_beschreibung := ' ';
		zyl_rafo_kamm.fb.st_config.str_instanz_name := 'Rasterfolien Kamm';
		zyl_rafo_kamm.fb.st_config.str_zylinder_typ := '2V2E_EIN_AUS';
		zyl_rafo_kamm.fb.st_config.t_ein_aus_fahrzeit := t#100ms;
		zyl_rafo_kamm.fb.st_config.t_ueberwachungszeit := t#1500ms;
		zyl_rafo_kamm.fb.st_config.i16_tzk_faktor_ausfahren := 100;
		zyl_rafo_kamm.fb.st_config.i16_tzk_faktor_einfahren := 100;
		zyl_rafo_kamm.fb.st_config.b_config_fertig := TRUE;

		(* Rasterfolien Vorzentrierer *)
		zyl_rafo_vorzentrierer.fb.st_config.b_config_fertig := FALSE;
		zyl_rafo_vorzentrierer.fb.st_config.b_endlage1_aktiv := TRUE;
		zyl_rafo_vorzentrierer.fb.st_config.b_endlage2_aktiv := FALSE;
		zyl_rafo_vorzentrierer.fb.st_config.b_sensor1_aktiv := TRUE;
		zyl_rafo_vorzentrierer.fb.st_config.b_sensor2_aktiv := FALSE;
		zyl_rafo_vorzentrierer.fb.st_config.i16_gruppe := 7;
		zyl_rafo_vorzentrierer.fb.st_config.i16_identnummer := 43;
		zyl_rafo_vorzentrierer.fb.st_config.i16_meld_startindex := 2840;
		zyl_rafo_vorzentrierer.fb.st_config.str_beschreibung := ' ';
		zyl_rafo_vorzentrierer.fb.st_config.str_instanz_name := 'Rasterfolien Vorzentrierer';
		zyl_rafo_vorzentrierer.fb.st_config.str_zylinder_typ := '2V2E_EIN_AUS';
		zyl_rafo_vorzentrierer.fb.st_config.t_ein_aus_fahrzeit := t#100ms;
		zyl_rafo_vorzentrierer.fb.st_config.t_ueberwachungszeit := t#1500ms;
		zyl_rafo_vorzentrierer.fb.st_config.i16_tzk_faktor_ausfahren := 100;
		zyl_rafo_vorzentrierer.fb.st_config.i16_tzk_faktor_einfahren := 100;
		zyl_rafo_vorzentrierer.fb.st_config.b_config_fertig := TRUE;

		(* Indexierzylinder Bestückposition *)
		zyl_Indexier_Bestueckpos.fb.st_config.b_config_fertig := FALSE;
		zyl_Indexier_Bestueckpos.fb.st_config.b_endlage1_aktiv := FALSE;
		zyl_Indexier_Bestueckpos.fb.st_config.b_endlage2_aktiv := FALSE;
		zyl_Indexier_Bestueckpos.fb.st_config.b_sensor1_aktiv := TRUE;
		zyl_Indexier_Bestueckpos.fb.st_config.b_sensor2_aktiv := TRUE;
		zyl_Indexier_Bestueckpos.fb.st_config.i16_gruppe := 3;
		zyl_Indexier_Bestueckpos.fb.st_config.i16_identnummer := 48;
		zyl_Indexier_Bestueckpos.fb.st_config.i16_meld_startindex := 2920;
		zyl_Indexier_Bestueckpos.fb.st_config.str_beschreibung := ' ';
		zyl_Indexier_Bestueckpos.fb.st_config.str_instanz_name := 'Indexierzylinder Bestückposition';
		zyl_Indexier_Bestueckpos.fb.st_config.str_zylinder_typ := '1V2E_EIN_AUS';
		zyl_Indexier_Bestueckpos.fb.st_config.t_ein_aus_fahrzeit := t#0ms;
		zyl_Indexier_Bestueckpos.fb.st_config.t_ueberwachungszeit := t#1000ms;
		zyl_Indexier_Bestueckpos.fb.st_config.i16_tzk_faktor_ausfahren := 100;
		zyl_Indexier_Bestueckpos.fb.st_config.i16_tzk_faktor_einfahren := 100;
		zyl_Indexier_Bestueckpos.fb.st_config.b_config_fertig := TRUE;

		(* Indexierzylinder Einlauf *)
		zyl_Indexier_Einlauf.fb.st_config.b_config_fertig := FALSE;
		zyl_Indexier_Einlauf.fb.st_config.b_endlage1_aktiv := FALSE;
		zyl_Indexier_Einlauf.fb.st_config.b_endlage2_aktiv := FALSE;
		zyl_Indexier_Einlauf.fb.st_config.b_sensor1_aktiv := TRUE;
		zyl_Indexier_Einlauf.fb.st_config.b_sensor2_aktiv := TRUE;
		zyl_Indexier_Einlauf.fb.st_config.i16_gruppe := 3;
		zyl_Indexier_Einlauf.fb.st_config.i16_identnummer := 49;
		zyl_Indexier_Einlauf.fb.st_config.i16_meld_startindex := 2940;
		zyl_Indexier_Einlauf.fb.st_config.str_beschreibung := ' ';
		zyl_Indexier_Einlauf.fb.st_config.str_instanz_name := ' Indexierzylinder Einlauf ';
		zyl_Indexier_Einlauf.fb.st_config.str_zylinder_typ := '1V2E_EIN_AUS';
		zyl_Indexier_Einlauf.fb.st_config.t_ein_aus_fahrzeit := t#0ms;
		zyl_Indexier_Einlauf.fb.st_config.t_ueberwachungszeit := t#1000ms;
		zyl_Indexier_Einlauf.fb.st_config.i16_tzk_faktor_ausfahren := 100;
		zyl_Indexier_Einlauf.fb.st_config.i16_tzk_faktor_einfahren := 100;
		zyl_Indexier_Einlauf.fb.st_config.b_config_fertig := TRUE;
ELSE
	b_config_fertig := FALSE;
END_IF
END_PROGRAM

(* POU Gemeinsamkeiten17xx/Oeler/ST_BandoelerZylinder, ST *)
PROGRAM ST_BandoelerZylinder
VAR_INPUT
	st_config						: struct_config;
	st_ctrl_in						: struct_ctrl_in;
	lr_achse_position				: LREAL;
	e_steuerung_ein				: BOOL;
	e_druckwaechter				: BOOL;

END_VAR
(*VAR_IN_OUT
	st_visu						: struct_oeler_visu;
END_VAR*)
VAR_OUTPUT
	st_ctrl_out					: struct_ctrl_out;
	b_oelmangel					: BOOL;
	st_oelerdaten					: struct_oeler_daten;
END_VAR
VAR
	fb_ton_uez					: TON;
	fb_ton_uez_fuellstand			: TON;
	fb_ton_quitt					: TON;
	fb_ton_speichern			: TON;
	fb_state_entry				: ST_StateEntry;
	fb_winkeltrigger				: ST_Winkeltrigger;
	b_hand_dialog_aktiv			: BOOL := FALSE;
	a_ventil_oben			 			AT %Q* : BOOL;
	a_ventil_unten			 			AT %Q* : BOOL;
	e_fuellstand					AT %I* : BOOL;
	e_druck_oelbehaelter			AT %I* : BOOL;
	sm_fuellstand_oeler			: BOOL := FALSE;
	sm_druckueberwachung		: BOOL := FALSE;
	bm_fuellstand_oeler			: BOOL := FALSE;
	b_ibn_handoelen				: BOOL := FALSE;
	fb_betriebsartenwechsel		: ST_Betriebsartenwechsel;
	fb_r_trig_bestueckhub			: R_TRIG;
	i16_hubzaehler				: INT := 0;
	fb_ton_oelen					: TON;
	b_zyl_unten					: BOOL;
	b_zyl_oben					: BOOL;
	dt_datum_uhrzeit_letzte_oelung	: DT;
	t_delta_zeitraum				: TIME := t#5h;
	fb_ton_oelzeit					: TON;
END_VAR
(*Mindestwerte eintragen damit nicht trocken gefahren werden kann*)
fb_ton_speichern(IN:= gst_datensatz.st_wkz.st_oeler.t_ventiloeffnungszeit<500 OR gst_datensatz.st_wkz.st_oeler.i16_intervall_bandoelen<1, PT:= t#20ms, Q=> , ET=> );
IF	fb_ton_speichern.Q THEN
	IF	gst_datensatz.st_wkz.st_oeler.t_ventiloeffnungszeit<50 THEN
		gst_datensatz.st_wkz.st_oeler.t_ventiloeffnungszeit:=500;
	END_IF

	IF	gst_datensatz.st_wkz.st_oeler.i16_intervall_bandoelen<1 THEN
		gst_datensatz.st_wkz.st_oeler.i16_intervall_bandoelen:=0;
	END_IF
END_IF

(* Bandöler mit Füllstandsabfrage *)
fb_ton_quitt(IN:= , PT:= t#100ms, Q=> , ET=> );
fb_ton_uez(IN:= NOT e_druck_oelbehaelter AND e_druckwaechter, PT:= t#60s, Q=> , ET=> );
fb_ton_uez_fuellstand(IN:= bm_fuellstand_oeler, PT:= t#1h, Q=> , ET=> );
fb_ton_oelen(IN:= , PT:= , Q=> , ET=> );

IF fb_state_entry.i16_step >= BEREIT AND fb_state_entry.i16_step < FEHLER THEN
	fb_winkeltrigger(IN:= LREAL_TO_INT(lr_achse_position), PT:= T#300ms, Q=> );
END_IF

(* Flanken *)
fb_r_trig_bestueckhub(CLK:= (gi16_betriebsart = AUTO OR gi16_betriebsart = TIPPEN) AND nockenschaltwerk_bestueckachse.fb.arr_spur[SP_OT], Q=> );

(* Hubzähler wird durch Nocke OT erhöht >> wenn der Zähler größer gleich dem Intervall ist wird a_ventil gesetzt *)
IF fb_r_trig_bestueckhub.Q THEN
	i16_hubzaehler := i16_hubzaehler + 1;
END_IF


(* Bandöler von Hand betätigen *)
IF gi16_betriebsart = HAND THEN
	a_ventil_oben :=  b_ibn_handoelen OR visu.b_handoelen ;
	a_ventil_unten :=  b_ibn_handoelen OR visu.b_handoelen ;
END_IF


(* Allgemeine Fehler *)

IF zyl_oelen_unten.st_ctrl.out.b_fehler OR
	zyl_oelen_oben.st_ctrl.out.b_fehler THEN
	fb_state_entry.i16_next_step := FEHLER;
END_IF

fb_betriebsartenwechsel(
	i16_akt_betriebsart:= gi16_betriebsart,
	b_wechsel_auto=> , 
	b_wechsel_tippen=> ,
	b_wechsel_hand=> , 
	b_wechsel_dummy=> , 
	b_wechsel_pseudo=> , 
	b_wechsel_allgemein=> );
(*
IF fb_betriebsartenwechsel.b_merker_ba_auto OR fb_betriebsartenwechsel.b_merker_ba_tippen THEN
	a_ventil := FALSE;
END_IF
*)

(* =======================================Toplevel========================================== *)
IF fb_state_entry.i16_next_step > INIT AND fb_state_entry.i16_next_step < FEHLER THEN
	IF fb_state_entry.i16_next_step < STOP THEN
		IF st_ctrl_in.b_stop THEN
			fb_state_entry.i16_next_step := STOP;
		END_IF
	END_IF
END_IF

(* Orangene Lampe an Ampel leuchtet bei Ölbehälter leer *)
b_oelmangel := bm_fuellstand_oeler;

(* ==================================Schrittkette================================ *)
fb_state_entry(
	i16_next_step:= , 
	i16_pos:= 1,
	s_debugtext:= ,
	E=> ,
	X=> ,
	i16_step=> ,
	i16_last_step=> );

CASE fb_state_entry.i16_step OF
(*=======================================================*)
	INIT_OBJ:
		IF st_config.b_config_fertig THEN
			fb_state_entry.i16_next_step := INIT;
		END_IF
		
(*=======================================================*)
	INIT:
		IF fb_state_entry.E THEN
			st_ctrl_out.b_fehler := FALSE;
			st_ctrl_out.b_bereit := FALSE;
			st_ctrl_out.b_fertig := FALSE;
			fb_ton_quitt.IN := FALSE;
			fb_ton_uez_fuellstand.IN := FALSE;
			a_ventil_oben := FALSE;
			a_ventil_unten := FALSE;
			sm_fuellstand_oeler := FALSE;
			sm_druckueberwachung := FALSE;
			bm_fuellstand_oeler := FALSE;
			st_ctrl_out.b_einzelfertigung := FALSE;
			fb_ton_oelen.IN := FALSE;
			b_zyl_unten:= FALSE;
			b_zyl_oben:= FALSE;
		END_IF

		(*-----------------------Weiterschaltbedingungen----------------------------*)
		IF st_ctrl_in.b_init THEN
			zyl_oelen_oben.st_ctrl.in.b_quittieren := FALSE;
			zyl_oelen_unten.st_ctrl.in.b_quittieren := FALSE;
			fb_state_entry.i16_next_step := 20;
		END_IF

(*=======================================================*)
	20: (* Abfrage Datum / Uhrzeit wegen Ölen nach Stillstand*)

		(*-----------------------Weiterschaltbedingungen----------------------------*)
		IF (gdt_system_time - dt_datum_uhrzeit_letzte_oelung) > t_delta_zeitraum THEN
			fb_ton_oelzeit.PT := st_oelerdaten.t_oelzeit_nach_stillstand;
			fb_state_entry.i16_next_step := 30;
		ELSE
			fb_state_entry.i16_next_step := BEREIT;
		END_IF

(*=======================================================*)
	30: (* Ölen nach Stillstand *)
		IF fb_state_entry.E THEN
			dt_datum_uhrzeit_letzte_oelung := gdt_system_time;	(* Merken, dass geölt wurde *)
			fb_ton_oelzeit.IN := TRUE;
			a_ventil_oben := TRUE;
			a_ventil_unten := TRUE;
		END_IF

		(*-----------------------Weiterschaltbedingungen----------------------------*)
		IF  fb_ton_oelzeit.Q THEN
			fb_ton_oelzeit.IN := FALSE;
			a_ventil_oben := FALSE;
			a_ventil_unten := FALSE;
			fb_state_entry.i16_next_step := BEREIT;
		END_IF

(*=======================================================
	40: (* Bandölen, abhängig von WKZ-Daten Zylinder ausfahren *)


	(*-----------------------Weiterschaltbedingungen----------------------------*)
		IF zyl_oelen_unten.fb.e_sensor1_ausgefahren AND
			 zyl_oelen_oben.fb.e_sensor1_ausgefahren THEN
			b_zyl_unten:= FALSE;
			b_zyl_oben:= FALSE;
			fb_state_entry.i16_next_step := 50;
		END_IF

(*=======================================================*)
	50: (* Bandölen, abhängig von WKZ-Daten Zylinder ausfahren *)


	(*-----------------------Weiterschaltbedingungen----------------------------*)
		IF zyl_oelen_unten.fb.e_sensor1_eingefahren AND
			 zyl_oelen_oben.fb.e_sensor1_eingefahren THEN
			fb_state_entry.i16_next_step := BEREIT;
		END_IF
=======================================================*)
	BEREIT:
		IF fb_state_entry.E THEN
			st_ctrl_out.b_bereit := TRUE;
		END_IF

		IF st_config.b_station_aktiv THEN
			(* Ölen *)
		(*	IF (gi16_betriebsart = AUTO OR gi16_betriebsart = TIPPEN) THEN
				IF	gst_datensatz.st_wkz.st_oeler.i16_intervall_bandoelen =0 THEN  (*bei Intervall 0 Dauerölen*)
					a_ventil_oben :=  fb_winkeltrigger.Q OR visu.b_handoelen OR b_ibn_handoelen;
					a_ventil_unten :=  fb_winkeltrigger.Q OR visu.b_handoelen OR b_ibn_handoelen;
				ELSE
					a_ventil_oben :=  visu.b_handoelen OR b_ibn_handoelen;
					a_ventil_unten :=  visu.b_handoelen OR b_ibn_handoelen;
				END_IF
			END_IF *)
			(* Überwachung Füllstand Betriebsmeldung*)
			IF NOT e_fuellstand AND e_steuerung_ein THEN
				bm_fuellstand_oeler := TRUE;
			ELSE
				bm_fuellstand_oeler := FALSE;
			END_IF
			(* Überwachung Füllstand Störmeldung *)
			IF fb_ton_uez_fuellstand.Q OR sm_fuellstand_oeler THEN
				sm_fuellstand_oeler := TRUE;
				st_ctrl_out.b_einzelfertigung:=TRUE;

				IF 	gi16_maschinenstatusinfo = STATUS_BETRIEBSBEREIT THEN
					fb_state_entry.i16_next_step := FEHLER;
				END_IF

			END_IF
			(* Überwachung Druck im Ölbehälter *)
			IF fb_ton_uez.Q OR sm_druckueberwachung THEN
				sm_druckueberwachung := TRUE;
				st_ctrl_out.b_einzelfertigung:=TRUE;

				IF 	gi16_maschinenstatusinfo = STATUS_BETRIEBSBEREIT THEN
					fb_state_entry.i16_next_step := FEHLER;
				END_IF
			END_IF

			(*-----------------------Weiterschaltbedingungen----------------------------*)
			IF	 i16_hubzaehler >= gst_datensatz.st_wkz.st_oeler.i16_intervall_bandoelen AND
				gst_datensatz.st_wkz.st_oeler.i16_intervall_bandoelen <>0 THEN (*bei Intervall 0 Dauerölen*)
				fb_state_entry.i16_next_step := 110;
			END_IF

		END_IF

(*=======================================================*)
	110: (* Bandölen, abhängig von WKZ-Daten Zylinder ausfahren *)
		IF fb_state_entry.E THEN
			dt_datum_uhrzeit_letzte_oelung := gdt_system_time;	(* Merken wann das letze mal geölt wurde *)
			i16_hubzaehler := 0;
			fb_ton_oelen.IN := TRUE;
			fb_ton_oelen.PT := DINT_TO_TIME(gst_datensatz.st_wkz.st_oeler.t_ventiloeffnungszeit);
			a_ventil_oben:= TRUE;
			a_ventil_unten:= TRUE;
		END_IF

		(*-----------------------Weiterschaltbedingungen----------------------------*)
		IF fb_ton_oelen.Q THEN
			fb_ton_oelen.IN := FALSE;
			a_ventil_oben := FALSE;
			a_ventil_unten := FALSE;
			fb_state_entry.i16_next_step := BEREIT;
		END_IF
(*=======================================================
	120: (* Bandölen, abhängig von WKZ-Daten Zylinder ausfahren *)


	(*-----------------------Weiterschaltbedingungen----------------------------*)
		IF zyl_oelen_unten.fb.e_sensor1_ausgefahren AND
			 zyl_oelen_oben.fb.e_sensor1_ausgefahren THEN
			b_zyl_unten:= FALSE;
			b_zyl_oben:= FALSE;
			fb_state_entry.i16_next_step := 130;
		END_IF

(*=======================================================*)
	130: (* Bandölen, abhängig von WKZ-Daten Zylinder ausfahren *)


	(*-----------------------Weiterschaltbedingungen----------------------------*)
		IF zyl_oelen_unten.fb.e_sensor1_eingefahren AND
			 zyl_oelen_oben.fb.e_sensor1_eingefahren THEN
			fb_state_entry.i16_next_step := BEREIT;
		END_IF
=======================================================*)
	FEHLER:
		IF fb_state_entry.E THEN
			st_ctrl_out.b_fehler := TRUE;
			a_ventil_oben := FALSE;
			a_ventil_unten := FALSE;
			fb_ton_quitt.IN := FALSE;
			zyl_oelen_oben.st_ctrl.in.b_quittieren := FALSE;
			zyl_oelen_unten.st_ctrl.in.b_quittieren := FALSE;
		END_IF

		(*-----------------------Weiterschaltbedingungen----------------------------*)
		IF st_ctrl_in.b_quitt AND NOT fb_state_entry.E THEN
			st_ctrl_out.b_fehler := FALSE;
			fb_ton_quitt.IN := TRUE;
			zyl_oelen_oben.st_ctrl.in.b_quittieren := TRUE;
			zyl_oelen_unten.st_ctrl.in.b_quittieren := TRUE;
		END_IF

		IF fb_ton_quitt.Q THEN
			fb_ton_quitt.IN := FALSE;
			fb_state_entry.i16_next_step := INIT;
		END_IF

(*=======================================================*)
	STOP:
		IF fb_state_entry.E THEN
			a_ventil_oben := FALSE;
			a_ventil_unten := FALSE;
			fb_ton_quitt.IN := FALSE;
			zyl_oelen_oben.st_ctrl.in.b_quittieren := FALSE;
			zyl_oelen_unten.st_ctrl.in.b_quittieren := FALSE;
		END_IF

		(*-----------------------Weiterschaltbedingungen----------------------------*)
		IF st_ctrl_in.b_quitt AND NOT fb_state_entry.E THEN
			fb_ton_quitt.IN := TRUE;
			zyl_oelen_oben.st_ctrl.in.b_quittieren := TRUE;
			zyl_oelen_unten.st_ctrl.in.b_quittieren := TRUE;
		END_IF

		IF fb_ton_quitt.Q THEN
			fb_ton_quitt.IN := FALSE;
			fb_state_entry.i16_next_step := INIT;
		END_IF
END_CASE

fb_state_entry(
	i16_next_step:= , 
	i16_pos:= 2,
	s_debugtext:= ,
	E=> ,
	X=> , 
	i16_step=> ,
	i16_last_step=> );

IF st_config.b_config_fertig THEN
	(* Fehlermeldungen und Betriebsmeldungen ab dem Startindex in die globalen Meldungsarrays schreiben *)
	garr_stoermeldungen[st_config.i16_meld_startindex + 0] := sm_fuellstand_oeler;
	garr_stoermeldungen[st_config.i16_meld_startindex + 1] := sm_druckueberwachung;
	garr_stoermeldungen[st_config.i16_meld_startindex + 2] := FALSE;
	garr_stoermeldungen[st_config.i16_meld_startindex + 3] := FALSE;
	garr_stoermeldungen[st_config.i16_meld_startindex + 4] := FALSE;
	garr_stoermeldungen[st_config.i16_meld_startindex + 5] := FALSE;
	garr_stoermeldungen[st_config.i16_meld_startindex + 6] := FALSE;
	garr_stoermeldungen[st_config.i16_meld_startindex + 7] := FALSE;
	garr_stoermeldungen[st_config.i16_meld_startindex + 8] := FALSE;
	garr_stoermeldungen[st_config.i16_meld_startindex + 9] := FALSE;
	garr_stoermeldungen[st_config.i16_meld_startindex + 10] := FALSE;
	garr_stoermeldungen[st_config.i16_meld_startindex + 11] := FALSE;
	garr_stoermeldungen[st_config.i16_meld_startindex + 12] := FALSE;
	garr_stoermeldungen[st_config.i16_meld_startindex + 13] := FALSE;
	garr_stoermeldungen[st_config.i16_meld_startindex + 14] := FALSE;
	garr_stoermeldungen[st_config.i16_meld_startindex + 15] := FALSE;
	garr_stoermeldungen[st_config.i16_meld_startindex + 16] := FALSE;
	garr_stoermeldungen[st_config.i16_meld_startindex + 17] := FALSE;
	garr_stoermeldungen[st_config.i16_meld_startindex + 18] := FALSE;
	garr_stoermeldungen[st_config.i16_meld_startindex + 19] := FALSE;
	
	garr_betriebsmeldungen[st_config.i16_meld_startindex + 0] := bm_fuellstand_oeler;
	garr_betriebsmeldungen[st_config.i16_meld_startindex + 1] := FALSE;
	garr_betriebsmeldungen[st_config.i16_meld_startindex + 2] := FALSE;
	garr_betriebsmeldungen[st_config.i16_meld_startindex + 3] := FALSE;
	garr_betriebsmeldungen[st_config.i16_meld_startindex + 4] := FALSE;
	garr_betriebsmeldungen[st_config.i16_meld_startindex + 5] := FALSE;
	garr_betriebsmeldungen[st_config.i16_meld_startindex + 6] := FALSE;
	garr_betriebsmeldungen[st_config.i16_meld_startindex + 7] := FALSE;
	garr_betriebsmeldungen[st_config.i16_meld_startindex + 8] := FALSE;
	garr_betriebsmeldungen[st_config.i16_meld_startindex + 9] := FALSE;
	garr_betriebsmeldungen[st_config.i16_meld_startindex + 10] := FALSE;
	garr_betriebsmeldungen[st_config.i16_meld_startindex + 11] := FALSE;
	garr_betriebsmeldungen[st_config.i16_meld_startindex + 12] := FALSE;
	garr_betriebsmeldungen[st_config.i16_meld_startindex + 13] := FALSE;
	garr_betriebsmeldungen[st_config.i16_meld_startindex + 14] := FALSE;
	garr_betriebsmeldungen[st_config.i16_meld_startindex + 15] := FALSE;
	garr_betriebsmeldungen[st_config.i16_meld_startindex + 16] := FALSE;
	garr_betriebsmeldungen[st_config.i16_meld_startindex + 17] := FALSE;
	garr_betriebsmeldungen[st_config.i16_meld_startindex + 18] := FALSE;
	garr_betriebsmeldungen[st_config.i16_meld_startindex + 19] := FALSE;
END_IF
END_PROGRAM

(* POU EPT Lib/Funktionsbausteine/ST_Winkeltrigger, ST *)
FUNCTION_BLOCK ST_Winkeltrigger
VAR_INPUT
	IN							: DINT;
	PT							: TIME;
END_VAR
VAR_OUTPUT
	Q							: BOOL;
END_VAR
VAR
	i32_alter_winkel				: DINT := 0;
	i32_neuer_winkel				: DINT := 0;
	b_triggersignal_start			: BOOL := FALSE;
	fb_tof_triggersignal			: TOF;
	t_zeit						: TIME := t#0ms;
END_VAR
(* Sobald sich der Hauptantrieb dreht, wird ein Triggersignal von mindestens 200ms erzeugt um Aktionen auszulösen *)
i32_neuer_winkel := IN;

IF PT < t#200ms THEN
	t_zeit := t#200ms;
ELSE
	t_zeit := PT;
END_IF

IF i32_neuer_winkel <> 360 THEN
	IF i32_neuer_winkel > i32_alter_winkel OR i32_neuer_winkel < i32_alter_winkel THEN
		b_triggersignal_start := TRUE;
	ELSE
		b_triggersignal_start := FALSE;
	END_IF
	i32_alter_winkel := i32_neuer_winkel;
ELSE
	b_triggersignal_start := FALSE;
END_IF

fb_tof_triggersignal(IN:= b_triggersignal_start, PT:= t_zeit, Q=> Q, ET=> );
END_FUNCTION_BLOCK

(* POU EPT Lib/Funktionsbausteine/ST_Betriebsartenwechsel, ST *)
FUNCTION_BLOCK ST_Betriebsartenwechsel
VAR_INPUT
	i16_akt_betriebsart		: enum_betriebsarten;
END_VAR
VAR_OUTPUT
	b_wechsel_auto			: BOOL;
	b_wechsel_tippen			: BOOL;
	b_wechsel_hand			: BOOL;
	b_wechsel_dummy		: BOOL;
	b_wechsel_pseudo		: BOOL;
	b_wechsel_allgemein		: BOOL;
END_VAR
VAR
	fb_r_trig_ba_auto			: R_TRIG;
	fb_r_trig_ba_tippen		: R_TRIG;
	fb_r_trig_ba_hand			: R_TRIG;
	fb_r_trig_ba_dummy		: R_TRIG;
	fb_r_trig_ba_pseudo		: R_TRIG;
	i16_betriebsart_alt			: enum_betriebsarten := KEINE;
	i16_betriebsart_neu		: enum_betriebsarten := KEINE;
	b_merker_ba_auto		: BOOL := FALSE;
	b_merker_ba_tippen		: BOOL := FALSE;
	b_merker_ba_hand		: BOOL := FALSE;
	b_merker_ba_dummy		: BOOL := FALSE;
	b_merker_ba_pseudo		: BOOL := FALSE;
END_VAR
(* Funktionsbaustein zum Erfassen der verschiedenen Betriebsartenflanken *)
fb_r_trig_ba_auto(CLK:= b_merker_ba_auto, Q=> b_wechsel_auto);
fb_r_trig_ba_tippen(CLK:= b_merker_ba_tippen, Q=> b_wechsel_tippen);
fb_r_trig_ba_hand(CLK:=b_merker_ba_hand , Q=> b_wechsel_hand);
fb_r_trig_ba_dummy(CLK:=b_merker_ba_dummy , Q=> b_wechsel_dummy);
fb_r_trig_ba_pseudo(CLK:=b_merker_ba_pseudo , Q=> b_wechsel_pseudo);

b_wechsel_allgemein := b_wechsel_auto OR b_wechsel_tippen OR b_wechsel_hand OR b_wechsel_dummy OR b_wechsel_pseudo;

i16_betriebsart_neu := i16_akt_betriebsart;

IF i16_betriebsart_neu <> i16_betriebsart_alt THEN
	CASE gi16_betriebsart OF
		KEINE:
			b_merker_ba_auto := FALSE;
			b_merker_ba_tippen := FALSE;
			b_merker_ba_hand := FALSE;
			b_merker_ba_dummy := FALSE;
			b_merker_ba_pseudo := FALSE;

		AUTO:
			b_merker_ba_auto := TRUE;
			b_merker_ba_tippen := FALSE;
			b_merker_ba_hand := FALSE;
			b_merker_ba_dummy := FALSE;
			b_merker_ba_pseudo := FALSE;

		TIPPEN:
			b_merker_ba_auto := FALSE;
			b_merker_ba_tippen := TRUE;
			b_merker_ba_hand := FALSE;
			b_merker_ba_dummy := FALSE;
			b_merker_ba_pseudo := FALSE;

		HAND:
			b_merker_ba_auto := FALSE;
			b_merker_ba_tippen := FALSE;
			b_merker_ba_hand := TRUE;
			b_merker_ba_dummy := FALSE;
			b_merker_ba_pseudo := FALSE;

		DUMMY:
			b_merker_ba_auto := FALSE;
			b_merker_ba_tippen := FALSE;
			b_merker_ba_hand := FALSE;
			b_merker_ba_dummy := TRUE;
			b_merker_ba_pseudo := FALSE;

		PSEUDO:
			b_merker_ba_auto := FALSE;
			b_merker_ba_tippen := FALSE;
			b_merker_ba_hand := FALSE;
			b_merker_ba_dummy := FALSE;
			b_merker_ba_pseudo := TRUE;
	END_CASE

	i16_betriebsart_alt := i16_betriebsart_neu;
END_IF
END_FUNCTION_BLOCK

(* POU Gemeinsamkeiten17xx/Oeler/ST_Doppelrollenbandoeler, ST *)
PROGRAM ST_Doppelrollenbandoeler
VAR_INPUT
	st_config						: struct_config;
	st_ctrl_in						: struct_ctrl_in;
	b_ot_spur					: BOOL;
END_VAR
VAR_IN_OUT
	st_visu						: struct_oeler_visu;
	st_oelerdaten					: struct_oeler_daten;
END_VAR
VAR_OUTPUT
	st_ctrl_out					: struct_ctrl_out;
	b_oelmangel					: BOOL;
END_VAR
VAR
	fb_ton_quitt					: TON;
	dt_datum_uhrzeit_letzte_oelung	: DT;
	fb_state_entry					: ST_StateEntry;
	t_delta_zeitraum				: TIME := t#5h;
	sm_fuellstand_oeler			: BOOL := FALSE;
	fb_ton_oelzeit					: TON;
	fb_r_trig_start_oelen			: R_TRIG;
	fb_r_trig_hubimpuls			: R_TRIG;
	b_ibn_handoelen				: BOOL := FALSE;
	bm_fuellstand_oeler			: BOOL := FALSE;
	a_ventil_rolle_li	 			AT %Q* : BOOL;
	a_ventil_rolle_re	 			AT %Q* : BOOL;
	e_fuellstand					AT %I* : BOOL;
END_VAR
(* Bandöler mit Füllstandsabfrage und Zwangs- und Stillstandsölung *)
(* Oeler Impuls generieren *)
fb_ton_oelzeit(IN:= , PT:= , Q=> , ET=> );
fb_ton_quitt(IN:= , PT:= t#100ms, Q=> , ET=> );

(* Hubimpuls *)
fb_r_trig_hubimpuls(CLK:= b_ot_spur, Q=> );

(* =======================================Toplevel========================================== *)
IF fb_state_entry.i16_next_step > INIT AND fb_state_entry.i16_next_step < FEHLER THEN
	IF fb_state_entry.i16_next_step < STOP THEN
		IF st_ctrl_in.b_stop THEN
			fb_state_entry.i16_next_step := STOP;
		END_IF
	END_IF
END_IF

(* Orangene Lampe an Ampel leuchtet bei Ölbehälter leer *)
b_oelmangel := bm_fuellstand_oeler;

(* =======================================Toplevel========================================== *)
IF fb_state_entry.i16_next_step > INIT AND fb_state_entry.i16_next_step < FEHLER THEN
	IF fb_state_entry.i16_next_step < STOP THEN
		IF st_ctrl_in.b_stop THEN
			fb_state_entry.i16_next_step := STOP;
		END_IF
	END_IF
END_IF

(* Prüfe auf neue Intervalvorgabe *)
IF st_config.b_station_aktiv AND st_oelerdaten.i32_neue_intervallvorgabe <> st_oelerdaten.i32_alte_intervallvorgabe THEN
	st_oelerdaten.i32_alte_intervallvorgabe := st_oelerdaten.i32_neue_intervallvorgabe;
	st_oelerdaten.i32_aktueller_stand := st_oelerdaten.i32_neue_intervallvorgabe;
END_IF

(* ==================================Schrittkette================================ *)
fb_state_entry(
	i16_next_step:= , 
	i16_pos:= 1,
	s_debugtext:= ,
	E=> ,
	X=> , 
	i16_step=> ,
	i16_last_step=> );

CASE fb_state_entry.i16_step OF
(*=======================================================*)
	INIT_OBJ:
		IF st_config.b_config_fertig THEN
			fb_state_entry.i16_next_step := INIT;
		END_IF
		
(*=======================================================*)
	INIT:
		IF fb_state_entry.E THEN
			st_ctrl_out.b_fehler := FALSE;
			st_ctrl_out.b_bereit := FALSE;
			st_ctrl_out.b_fertig := FALSE;
			fb_ton_oelzeit.IN := FALSE;
			fb_ton_quitt.IN := FALSE;
			a_ventil_rolle_li := FALSE;
			a_ventil_rolle_re := FALSE;
			sm_fuellstand_oeler := FALSE;
			bm_fuellstand_oeler := FALSE;
		END_IF

		(*-----------------------Weiterschaltbedingungen----------------------------*)
		IF st_ctrl_in.b_init THEN
			IF st_config.b_station_aktiv THEN
				fb_state_entry.i16_next_step := 20;
			ELSE
				fb_state_entry.i16_next_step := BEREIT;
			END_IF
		END_IF

(*=======================================================*)
	20: (* Abfrage Datum / Uhrzeit wegen Ölen nach Stillstand*)

		(*-----------------------Weiterschaltbedingungen----------------------------*)
		IF (gdt_system_time - dt_datum_uhrzeit_letzte_oelung) > t_delta_zeitraum THEN
			fb_ton_oelzeit.PT := st_oelerdaten.t_oelzeit_nach_stillstand;
			fb_state_entry.i16_next_step := 30;
		ELSE
			fb_state_entry.i16_next_step := BEREIT;
		END_IF

(*=======================================================*)
	30: (* Ölen nach Stillstand *)
		IF fb_state_entry.E THEN
			dt_datum_uhrzeit_letzte_oelung := gdt_system_time;	(* Merken, dass geölt wurde *)
			fb_ton_oelzeit.IN := TRUE;
			a_ventil_rolle_li := TRUE;
			a_ventil_rolle_re := TRUE;
		END_IF

		(*-----------------------Weiterschaltbedingungen----------------------------*)
		IF  fb_ton_oelzeit.Q THEN
			fb_ton_oelzeit.IN := FALSE;
			a_ventil_rolle_li := FALSE;
			a_ventil_rolle_re := FALSE;
			fb_state_entry.i16_next_step := BEREIT;
		END_IF

(*=======================================================*)
	BEREIT:
		IF fb_state_entry.E THEN
			st_ctrl_out.b_bereit := TRUE;
		END_IF

		IF st_config.b_station_aktiv THEN
			(* Zähle Hübe *)
			IF fb_r_trig_hubimpuls.Q THEN
				(* Von der Intervallvorgabe wird runter gezählt bis Null. Dann kommt der Ölimpuls *)
				st_oelerdaten.i32_aktueller_stand := st_oelerdaten.i32_aktueller_stand - 1;
			END_IF
			(* Überwachung Füllstand *)
			IF NOT e_fuellstand THEN
				sm_fuellstand_oeler := TRUE;
				fb_state_entry.i16_next_step := FEHLER;
			END_IF

			(*-----------------------Weiterschaltbedingungen----------------------------*)
			IF  st_oelerdaten.i32_aktueller_stand <= 0 OR st_visu.b_handoelen OR b_ibn_handoelen THEN
				st_visu.b_handoelen := FALSE;
				fb_ton_oelzeit.PT := st_oelerdaten.t_ventiloeffnungszeit;
				fb_state_entry.i16_next_step := 110;
			END_IF
		END_IF

(*=======================================================*)
	110: (* Ölen *)
		IF fb_state_entry.E THEN
			dt_datum_uhrzeit_letzte_oelung := gdt_system_time;	(* Merken wann das letze mal geölt wurde *)
			IF st_oelerdaten.i32_neue_intervallvorgabe <= 0 THEN
				 st_oelerdaten.i32_neue_intervallvorgabe := 100;	(* Verhindere Dauerölung, wenn in den WKZ-Ölerdaten noch 0 drin steht *)
			END_IF
			st_oelerdaten.i32_aktueller_stand := st_oelerdaten.i32_neue_intervallvorgabe;
			fb_ton_oelzeit.IN := TRUE;
			a_ventil_rolle_li := TRUE;
			a_ventil_rolle_re := TRUE;
		END_IF

		(* Zähle Hübe *)
		IF fb_r_trig_hubimpuls.Q THEN
			(* Von der Intervallvorgabe wird runter gezählt bis Null. Dann kommt der Ölimpuls *)
			st_oelerdaten.i32_aktueller_stand := st_oelerdaten.i32_aktueller_stand - 1;
		END_IF

		(*-----------------------Weiterschaltbedingungen----------------------------*)
		IF  fb_ton_oelzeit.Q THEN
			fb_ton_oelzeit.IN := FALSE;
			a_ventil_rolle_li := FALSE;
			a_ventil_rolle_re := FALSE;
			fb_state_entry.i16_next_step := BEREIT;
		END_IF

(*=======================================================*)
	FEHLER:
		IF fb_state_entry.E THEN
			st_ctrl_out.b_fehler := TRUE;
			a_ventil_rolle_li := FALSE;
			a_ventil_rolle_re := FALSE;
			fb_ton_quitt.IN := FALSE;
		END_IF

		(*-----------------------Weiterschaltbedingungen----------------------------*)
		IF st_ctrl_in.b_quitt AND NOT fb_state_entry.E THEN
			st_ctrl_out.b_fehler := FALSE;
			fb_ton_quitt.IN := TRUE;
		END_IF

		IF fb_ton_quitt.Q THEN
			fb_ton_quitt.IN := FALSE;
			fb_state_entry.i16_next_step := INIT;
		END_IF

(*=======================================================*)
	STOP:
		IF fb_state_entry.E THEN
			a_ventil_rolle_li := FALSE;
			a_ventil_rolle_re := FALSE;
			fb_ton_quitt.IN := FALSE;
		END_IF

		(*-----------------------Weiterschaltbedingungen----------------------------*)
		IF st_ctrl_in.b_quitt AND NOT fb_state_entry.E THEN
			fb_ton_quitt.IN := TRUE;
		END_IF

		IF fb_ton_quitt.Q THEN
			fb_ton_quitt.IN := FALSE;
			fb_state_entry.i16_next_step := INIT;
		END_IF
END_CASE

fb_state_entry(
	i16_next_step:= , 
	i16_pos:= 2,
	s_debugtext:= ,
	E=> ,
	X=> , 
	i16_step=> ,
	i16_last_step=> );

IF st_config.b_config_fertig THEN
	(* Fehlermeldungen und Betriebsmeldungen ab dem Startindex in die globalen Meldungsarrays schreiben *)
	garr_stoermeldungen[st_config.i16_meld_startindex + 0] := sm_fuellstand_oeler;
	garr_stoermeldungen[st_config.i16_meld_startindex + 1] := FALSE;
	garr_stoermeldungen[st_config.i16_meld_startindex + 2] := FALSE;
	garr_stoermeldungen[st_config.i16_meld_startindex + 3] := FALSE;
	garr_stoermeldungen[st_config.i16_meld_startindex + 4] := FALSE;
	garr_stoermeldungen[st_config.i16_meld_startindex + 5] := FALSE;
	garr_stoermeldungen[st_config.i16_meld_startindex + 6] := FALSE;
	garr_stoermeldungen[st_config.i16_meld_startindex + 7] := FALSE;
	garr_stoermeldungen[st_config.i16_meld_startindex + 8] := FALSE;
	garr_stoermeldungen[st_config.i16_meld_startindex + 9] := FALSE;
	garr_stoermeldungen[st_config.i16_meld_startindex + 10] := FALSE;
	garr_stoermeldungen[st_config.i16_meld_startindex + 11] := FALSE;
	garr_stoermeldungen[st_config.i16_meld_startindex + 12] := FALSE;
	garr_stoermeldungen[st_config.i16_meld_startindex + 13] := FALSE;
	garr_stoermeldungen[st_config.i16_meld_startindex + 14] := FALSE;
	garr_stoermeldungen[st_config.i16_meld_startindex + 15] := FALSE;
	garr_stoermeldungen[st_config.i16_meld_startindex + 16] := FALSE;
	garr_stoermeldungen[st_config.i16_meld_startindex + 17] := FALSE;
	garr_stoermeldungen[st_config.i16_meld_startindex + 18] := FALSE;
	garr_stoermeldungen[st_config.i16_meld_startindex + 19] := FALSE;
	
	garr_betriebsmeldungen[st_config.i16_meld_startindex + 0] := bm_fuellstand_oeler;
	garr_betriebsmeldungen[st_config.i16_meld_startindex + 1] := FALSE;
	garr_betriebsmeldungen[st_config.i16_meld_startindex + 2] := FALSE;
	garr_betriebsmeldungen[st_config.i16_meld_startindex + 3] := FALSE;
	garr_betriebsmeldungen[st_config.i16_meld_startindex + 4] := FALSE;
	garr_betriebsmeldungen[st_config.i16_meld_startindex + 5] := FALSE;
	garr_betriebsmeldungen[st_config.i16_meld_startindex + 6] := FALSE;
	garr_betriebsmeldungen[st_config.i16_meld_startindex + 7] := FALSE;
	garr_betriebsmeldungen[st_config.i16_meld_startindex + 8] := FALSE;
	garr_betriebsmeldungen[st_config.i16_meld_startindex + 9] := FALSE;
	garr_betriebsmeldungen[st_config.i16_meld_startindex + 10] := FALSE;
	garr_betriebsmeldungen[st_config.i16_meld_startindex + 11] := FALSE;
	garr_betriebsmeldungen[st_config.i16_meld_startindex + 12] := FALSE;
	garr_betriebsmeldungen[st_config.i16_meld_startindex + 13] := FALSE;
	garr_betriebsmeldungen[st_config.i16_meld_startindex + 14] := FALSE;
	garr_betriebsmeldungen[st_config.i16_meld_startindex + 15] := FALSE;
	garr_betriebsmeldungen[st_config.i16_meld_startindex + 16] := FALSE;
	garr_betriebsmeldungen[st_config.i16_meld_startindex + 17] := FALSE;
	garr_betriebsmeldungen[st_config.i16_meld_startindex + 18] := FALSE;
	garr_betriebsmeldungen[st_config.i16_meld_startindex + 19] := FALSE;
END_IF
END_PROGRAM

(* POU Gemeinsamkeiten17xx/Oeler/ST_Einzelbandoeler, ST *)
PROGRAM ST_Einzelbandoeler
VAR_INPUT
	st_config						: struct_config;
	st_ctrl_in						: struct_ctrl_in;
	b_ot_spur					: BOOL;
END_VAR
VAR_IN_OUT
	st_visu						: struct_oeler_visu;
	st_oelerdaten					: struct_oeler_retain;
END_VAR
VAR_OUTPUT
	st_ctrl_out					: struct_ctrl_out;
END_VAR
VAR
	fb_ton_quitt					: TON;
	dt_datum_uhrzeit_letzte_oelung	: DT;
	fb_state_entry					: ST_StateEntry;
	t_delta_zeitraum				: TIME := t#5h;
	a_ventil			 			AT %Q* : BOOL;
	e_fuellstand					AT %I* : BOOL;
	sm_fuellstand_oeler			: BOOL := FALSE;
	fb_ton_oelzeit					: TON;
	fb_r_trig_start_oelen			: R_TRIG;
	fb_r_trig_hubimpuls			: R_TRIG;

	fb_r_trig_ibn_handoelen		: R_TRIG;
	fb_ton_ibn_handoelen			: TON;
	b_ibn_handoelen				: BOOL := FALSE;
END_VAR
(* Bandöler mit Füllstandsabfrage und Zwangs- und Stillstandsölung *)
(* Oeler Impuls generieren *)
fb_ton_oelzeit(IN:= , PT:= , Q=> , ET=> );
fb_ton_quitt(IN:= , PT:= t#100ms, Q=> , ET=> );

(* Hubimpuls *)
fb_r_trig_hubimpuls(CLK:= b_ot_spur, Q=> );

(* Inbetriebnahme *)
fb_r_trig_ibn_handoelen(CLK:= b_ibn_handoelen, Q=> );
fb_ton_ibn_handoelen(IN:= , PT:= t#1s, Q=> , ET=> );
IF fb_r_trig_ibn_handoelen.Q THEN
	fb_ton_ibn_handoelen.IN := TRUE;
ELSE
	IF fb_ton_ibn_handoelen.Q THEN
		b_ibn_handoelen := FALSE;
	 	fb_ton_ibn_handoelen.IN := FALSE;
	END_IF
END_IF

(* =======================================Toplevel========================================== *)
IF fb_state_entry.i16_next_step > INIT AND fb_state_entry.i16_next_step < FEHLER THEN
	IF fb_state_entry.i16_next_step < STOP THEN
		IF st_ctrl_in.b_stop THEN
			fb_state_entry.i16_next_step := STOP;
		END_IF
	END_IF
END_IF

(* Prüfe auf neue Intervalvorgabe *)
IF st_config.b_station_aktiv AND st_oelerdaten.i32_neue_intervallvorgabe <> st_oelerdaten.i32_alte_intervallvorgabe THEN
	st_oelerdaten.i32_alte_intervallvorgabe := st_oelerdaten.i32_neue_intervallvorgabe;
	st_oelerdaten.i32_aktueller_stand := st_oelerdaten.i32_neue_intervallvorgabe;
END_IF

(* ==================================Schrittkette================================ *)
fb_state_entry(
	i16_next_step:= , 
	i16_pos:= 1,
	s_debugtext:= ,
	E=> ,
	X=> , 
	i16_step=> ,
	i16_last_step=> );

CASE fb_state_entry.i16_step OF
(*=======================================================*)
	INIT_OBJ:
		IF st_config.b_config_fertig THEN
			fb_state_entry.i16_next_step := INIT;
		END_IF
		
(*=======================================================*)
	INIT:
		IF fb_state_entry.E THEN
			st_ctrl_out.b_fehler := FALSE;
			st_ctrl_out.b_bereit := FALSE;
			st_ctrl_out.b_fertig := FALSE;
			fb_ton_oelzeit.IN := FALSE;
			fb_ton_ibn_handoelen.IN := FALSE;
			fb_ton_quitt.IN := FALSE;
			a_ventil := FALSE;
			sm_fuellstand_oeler := FALSE;
		END_IF

		(*-----------------------Weiterschaltbedingungen----------------------------*)
		IF st_ctrl_in.b_init THEN
			IF st_config.b_station_aktiv THEN
				fb_state_entry.i16_next_step := 20;
			ELSE
				fb_state_entry.i16_next_step := BEREIT;
			END_IF
		END_IF

(*=======================================================*)
	20: (* Abfrage Datum / Uhrzeit wegen Ölen nach Stillstand*)

		(*-----------------------Weiterschaltbedingungen----------------------------*)
		IF (gdt_system_time - dt_datum_uhrzeit_letzte_oelung) > t_delta_zeitraum THEN
			fb_ton_oelzeit.PT := st_oelerdaten.t_oelzeit_nach_stillstand;
			fb_state_entry.i16_next_step := 30;
		ELSE
			fb_state_entry.i16_next_step := BEREIT;
		END_IF

(*=======================================================*)
	30: (* Ölen nach Stillstand *)
		IF fb_state_entry.E THEN
			dt_datum_uhrzeit_letzte_oelung := gdt_system_time;	(* Merken, dass geölt wurde *)
			fb_ton_oelzeit.IN := TRUE;
			a_ventil := TRUE;
		END_IF

		(*-----------------------Weiterschaltbedingungen----------------------------*)
		IF  fb_ton_oelzeit.Q THEN
			fb_ton_oelzeit.IN := FALSE;
			a_ventil := FALSE;
			fb_state_entry.i16_next_step := BEREIT;
		END_IF

(*=======================================================*)
	BEREIT:
		IF fb_state_entry.E THEN
			st_ctrl_out.b_bereit := TRUE;
		END_IF

		IF st_config.b_station_aktiv THEN
			(* Zähle Hübe *)
			IF fb_r_trig_hubimpuls.Q THEN
				(* Von der Intervallvorgabe wird runter gezählt bis Null. Dann kommt der Ölimpuls *)
				st_oelerdaten.i32_aktueller_stand := st_oelerdaten.i32_aktueller_stand - 1;
			END_IF
			(* Überwachung Füllstand *)
			IF NOT e_fuellstand THEN
				sm_fuellstand_oeler := TRUE;
				fb_state_entry.i16_next_step := FEHLER;
			END_IF

			(*-----------------------Weiterschaltbedingungen----------------------------*)
			IF  st_oelerdaten.i32_aktueller_stand <= 0 OR st_visu.b_handoelen OR fb_r_trig_ibn_handoelen.Q THEN
				st_visu.b_handoelen := FALSE;
				fb_ton_oelzeit.PT := st_oelerdaten.t_ventiloeffnungszeit;
				fb_state_entry.i16_next_step := 110;
			END_IF
		END_IF

(*=======================================================*)
	110: (* Ölen *)
		IF fb_state_entry.E THEN
			dt_datum_uhrzeit_letzte_oelung := gdt_system_time;	(* Merken wann das letze mal geölt wurde *)
			IF st_oelerdaten.i32_neue_intervallvorgabe <= 0 THEN
				 st_oelerdaten.i32_neue_intervallvorgabe := 100;	(* Verhindere Dauerölung, wenn in den WKZ-Ölerdaten noch 0 drin steht *)
			END_IF
			st_oelerdaten.i32_aktueller_stand := st_oelerdaten.i32_neue_intervallvorgabe;
			fb_ton_oelzeit.IN := TRUE;
			a_ventil := TRUE;
		END_IF

		(* Zähle Hübe *)
		IF fb_r_trig_hubimpuls.Q THEN
			(* Von der Intervallvorgabe wird runter gezählt bis Null. Dann kommt der Ölimpuls *)
			st_oelerdaten.i32_aktueller_stand := st_oelerdaten.i32_aktueller_stand - 1;
		END_IF

		(*-----------------------Weiterschaltbedingungen----------------------------*)
		IF  fb_ton_oelzeit.Q THEN
			fb_ton_oelzeit.IN := FALSE;
			a_ventil := FALSE;
			fb_state_entry.i16_next_step := BEREIT;
		END_IF

(*=======================================================*)
	FEHLER:
		IF fb_state_entry.E THEN
			st_ctrl_out.b_fehler := TRUE;
			a_ventil := FALSE;
			fb_ton_quitt.IN := FALSE;
		END_IF

		(*-----------------------Weiterschaltbedingungen----------------------------*)
		IF st_ctrl_in.b_quitt AND NOT fb_state_entry.E THEN
			st_ctrl_out.b_fehler := FALSE;
			fb_ton_quitt.IN := TRUE;
		END_IF

		IF fb_ton_quitt.Q THEN
			fb_ton_quitt.IN := FALSE;
			fb_state_entry.i16_next_step := INIT;
		END_IF

(*=======================================================*)
	STOP:
		IF fb_state_entry.E THEN
			a_ventil := FALSE;
			fb_ton_quitt.IN := FALSE;
		END_IF

		(*-----------------------Weiterschaltbedingungen----------------------------*)
		IF st_ctrl_in.b_quitt AND NOT fb_state_entry.E THEN
			fb_ton_quitt.IN := TRUE;
		END_IF

		IF fb_ton_quitt.Q THEN
			fb_ton_quitt.IN := FALSE;
			fb_state_entry.i16_next_step := INIT;
		END_IF
END_CASE

fb_state_entry(
	i16_next_step:= , 
	i16_pos:= 2,
	s_debugtext:= ,
	E=> ,
	X=> , 
	i16_step=> ,
	i16_last_step=> );

IF st_config.b_config_fertig THEN
	(* Fehlermeldungen und Betriebsmeldungen ab dem Startindex in die globalen Meldungsarrays schreiben *)
	garr_stoermeldungen[st_config.i16_meld_startindex + 0] := sm_fuellstand_oeler;
	garr_stoermeldungen[st_config.i16_meld_startindex + 1] := FALSE;
	garr_stoermeldungen[st_config.i16_meld_startindex + 2] := FALSE;
	garr_stoermeldungen[st_config.i16_meld_startindex + 3] := FALSE;
	garr_stoermeldungen[st_config.i16_meld_startindex + 4] := FALSE;
	garr_stoermeldungen[st_config.i16_meld_startindex + 5] := FALSE;
	garr_stoermeldungen[st_config.i16_meld_startindex + 6] := FALSE;
	garr_stoermeldungen[st_config.i16_meld_startindex + 7] := FALSE;
	garr_stoermeldungen[st_config.i16_meld_startindex + 8] := FALSE;
	garr_stoermeldungen[st_config.i16_meld_startindex + 9] := FALSE;
	garr_stoermeldungen[st_config.i16_meld_startindex + 10] := FALSE;
	garr_stoermeldungen[st_config.i16_meld_startindex + 11] := FALSE;
	garr_stoermeldungen[st_config.i16_meld_startindex + 12] := FALSE;
	garr_stoermeldungen[st_config.i16_meld_startindex + 13] := FALSE;
	garr_stoermeldungen[st_config.i16_meld_startindex + 14] := FALSE;
	garr_stoermeldungen[st_config.i16_meld_startindex + 15] := FALSE;
	garr_stoermeldungen[st_config.i16_meld_startindex + 16] := FALSE;
	garr_stoermeldungen[st_config.i16_meld_startindex + 17] := FALSE;
	garr_stoermeldungen[st_config.i16_meld_startindex + 18] := FALSE;
	garr_stoermeldungen[st_config.i16_meld_startindex + 19] := FALSE;
	
	garr_betriebsmeldungen[st_config.i16_meld_startindex + 0] := FALSE;
	garr_betriebsmeldungen[st_config.i16_meld_startindex + 1] := FALSE;
	garr_betriebsmeldungen[st_config.i16_meld_startindex + 2] := FALSE;
	garr_betriebsmeldungen[st_config.i16_meld_startindex + 3] := FALSE;
	garr_betriebsmeldungen[st_config.i16_meld_startindex + 4] := FALSE;
	garr_betriebsmeldungen[st_config.i16_meld_startindex + 5] := FALSE;
	garr_betriebsmeldungen[st_config.i16_meld_startindex + 6] := FALSE;
	garr_betriebsmeldungen[st_config.i16_meld_startindex + 7] := FALSE;
	garr_betriebsmeldungen[st_config.i16_meld_startindex + 8] := FALSE;
	garr_betriebsmeldungen[st_config.i16_meld_startindex + 9] := FALSE;
	garr_betriebsmeldungen[st_config.i16_meld_startindex + 10] := FALSE;
	garr_betriebsmeldungen[st_config.i16_meld_startindex + 11] := FALSE;
	garr_betriebsmeldungen[st_config.i16_meld_startindex + 12] := FALSE;
	garr_betriebsmeldungen[st_config.i16_meld_startindex + 13] := FALSE;
	garr_betriebsmeldungen[st_config.i16_meld_startindex + 14] := FALSE;
	garr_betriebsmeldungen[st_config.i16_meld_startindex + 15] := FALSE;
	garr_betriebsmeldungen[st_config.i16_meld_startindex + 16] := FALSE;
	garr_betriebsmeldungen[st_config.i16_meld_startindex + 17] := FALSE;
	garr_betriebsmeldungen[st_config.i16_meld_startindex + 18] := FALSE;
	garr_betriebsmeldungen[st_config.i16_meld_startindex + 19] := FALSE;
END_IF
END_PROGRAM

(* POU Gemeinsamkeiten17xx/Oeler/ST_Menzel_Spruehoeler, ST *)
PROGRAM ST_Menzel_Spruehoeler
VAR_INPUT
	st_config						: struct_config;
	st_ctrl_in						: struct_ctrl_in;
	lr_achse_position				: LREAL;
	e_steuerung_ein				: BOOL;
	e_druckwaechter				: BOOL;
END_VAR
(*VAR_IN_OUT
	st_visu						: struct_oeler_visu;
END_VAR*)
VAR_OUTPUT
	st_ctrl_out					: struct_ctrl_out;
	b_oelmangel					: BOOL;
END_VAR
VAR
	fb_ton_uez					: TON;
	fb_ton_uez_fuellstand			: TON;
	fb_ton_quitt					: TON;
	fb_ton_speichern			: TON;
	fb_state_entry				: ST_StateEntry;
	fb_winkeltrigger				: ST_Winkeltrigger;
	b_hand_dialog_aktiv			: BOOL := FALSE;
	a_ventil			 			AT %Q* : BOOL;
	e_fuellstand					AT %I* : BOOL;
	e_druck_oelbehaelter			AT %I* : BOOL;
	sm_fuellstand_oeler			: BOOL := FALSE;
	sm_druckueberwachung		: BOOL := FALSE;
	bm_fuellstand_oeler			: BOOL := FALSE;
	b_ibn_handoelen				: BOOL := FALSE;
	fb_betriebsartenwechsel		: ST_Betriebsartenwechsel;
	fb_r_trig_bestueckhub			: R_TRIG;
	i16_hubzaehler				: INT := 0;
	fb_ton_oelen					: TON;
END_VAR
(*Intervalllölen wird beim Sprühöler nicht mehr benötigt, darum wird der Wert auf Null geforced*)
gst_datensatz.st_wkz.st_oeler.i16_intervall_bandoelen:=0;

(*Mindestwerte eintragen damit nicht trocken gefahren werden kann*)
fb_ton_speichern(IN:= gst_datensatz.st_wkz.st_oeler.t_ventiloeffnungszeit<500 OR gst_datensatz.st_wkz.st_oeler.i16_intervall_bandoelen<1, PT:= t#20ms, Q=> , ET=> );
IF	fb_ton_speichern.Q THEN
	IF	gst_datensatz.st_wkz.st_oeler.t_ventiloeffnungszeit<500 THEN
		gst_datensatz.st_wkz.st_oeler.t_ventiloeffnungszeit:=500;
	END_IF

	IF	gst_datensatz.st_wkz.st_oeler.i16_intervall_bandoelen<1 THEN
		gst_datensatz.st_wkz.st_oeler.i16_intervall_bandoelen:=0;
	END_IF
END_IF

(* Bandöler mit Füllstandsabfrage *)
fb_ton_quitt(IN:= , PT:= t#100ms, Q=> , ET=> );
fb_ton_uez(IN:= NOT e_druck_oelbehaelter AND e_druckwaechter, PT:= t#60s, Q=> , ET=> );
fb_ton_uez_fuellstand(IN:= bm_fuellstand_oeler, PT:= t#1h, Q=> , ET=> );
fb_ton_oelen(IN:= , PT:= , Q=> , ET=> );

IF fb_state_entry.i16_step >= BEREIT AND fb_state_entry.i16_step < FEHLER THEN
	fb_winkeltrigger(IN:= LREAL_TO_INT(lr_achse_position), PT:= T#300ms, Q=> );
END_IF

(* Flanken *)
fb_r_trig_bestueckhub(CLK:= (gi16_betriebsart = AUTO OR gi16_betriebsart = TIPPEN) AND nockenschaltwerk_bestueckachse.fb.arr_spur[SP_OT], Q=> );

(* Hubzähler wird durch Nocke OT erhöht >> wenn der Zähler größer gleich dem Intervall ist wird a_ventil gesetzt *)
IF fb_r_trig_bestueckhub.Q THEN
	i16_hubzaehler := i16_hubzaehler + 1;
END_IF

(* Bandöler von Hand betätigen *)
IF gi16_betriebsart = HAND THEN
	a_ventil :=  b_ibn_handoelen OR (b_hand_dialog_aktiv AND (visu.b_handoelen OR ST_Euchner_Handbedienpult.b_Taste_Power));
END_IF

fb_betriebsartenwechsel(
	i16_akt_betriebsart:= gi16_betriebsart,
	b_wechsel_auto=> , 
	b_wechsel_tippen=> ,
	b_wechsel_hand=> , 
	b_wechsel_dummy=> , 
	b_wechsel_pseudo=> , 
	b_wechsel_allgemein=> );
(*
IF fb_betriebsartenwechsel.b_merker_ba_auto OR fb_betriebsartenwechsel.b_merker_ba_tippen THEN
	a_ventil := FALSE;
END_IF
*)

(* =======================================Toplevel========================================== *)
IF fb_state_entry.i16_next_step > INIT AND fb_state_entry.i16_next_step < FEHLER THEN
	IF fb_state_entry.i16_next_step < STOP THEN
		IF st_ctrl_in.b_stop THEN
			fb_state_entry.i16_next_step := STOP;
		END_IF
	END_IF
END_IF

(* Orangene Lampe an Ampel leuchtet bei Ölbehälter leer *)
b_oelmangel := bm_fuellstand_oeler;

(* ==================================Schrittkette================================ *)
fb_state_entry(
	i16_next_step:= , 
	i16_pos:= 1,
	s_debugtext:= ,
	E=> ,
	X=> ,
	i16_step=> ,
	i16_last_step=> );

CASE fb_state_entry.i16_step OF
(*=======================================================*)
	INIT_OBJ:
		IF st_config.b_config_fertig THEN
			fb_state_entry.i16_next_step := INIT;
		END_IF
		
(*=======================================================*)
	INIT:
		IF fb_state_entry.E THEN
			st_ctrl_out.b_fehler := FALSE;
			st_ctrl_out.b_bereit := FALSE;
			st_ctrl_out.b_fertig := FALSE;
			fb_ton_quitt.IN := FALSE;
			fb_ton_uez_fuellstand.IN := FALSE;
			a_ventil := FALSE;
			sm_fuellstand_oeler := FALSE;
			sm_druckueberwachung := FALSE;
			bm_fuellstand_oeler := FALSE;
			st_ctrl_out.b_einzelfertigung := FALSE;
			fb_ton_oelen.IN := FALSE;
		END_IF

		(*-----------------------Weiterschaltbedingungen----------------------------*)
		IF st_ctrl_in.b_init THEN
			fb_state_entry.i16_next_step := BEREIT;
		END_IF

(*=======================================================*)
	BEREIT:
		IF fb_state_entry.E THEN
			st_ctrl_out.b_bereit := TRUE;
		END_IF

		IF st_config.b_station_aktiv THEN
			(* Ölen *)
			IF (gi16_betriebsart = AUTO OR gi16_betriebsart = TIPPEN) THEN
				IF	gst_datensatz.st_wkz.st_oeler.i16_intervall_bandoelen =0 THEN  (*bei Intervall 0 Dauerölen*)
					a_ventil :=  fb_winkeltrigger.Q OR visu.b_handoelen OR b_ibn_handoelen;
				ELSE
					a_ventil :=  visu.b_handoelen OR b_ibn_handoelen;
				END_IF
			END_IF
			(* Überwachung Füllstand Betriebsmeldung*)
			IF NOT e_fuellstand AND e_steuerung_ein THEN
				bm_fuellstand_oeler := TRUE;
			ELSE
				bm_fuellstand_oeler := FALSE;
			END_IF
			(* Überwachung Füllstand Störmeldung *)
			IF fb_ton_uez_fuellstand.Q OR sm_fuellstand_oeler THEN
				sm_fuellstand_oeler := TRUE;
				st_ctrl_out.b_einzelfertigung:=TRUE;

				IF 	gi16_maschinenstatusinfo = STATUS_BETRIEBSBEREIT THEN
					fb_state_entry.i16_next_step := FEHLER;
				END_IF

			END_IF
			(* Überwachung Druck im Ölbehälter *)
			IF fb_ton_uez.Q OR sm_druckueberwachung THEN
				sm_druckueberwachung := TRUE;
				st_ctrl_out.b_einzelfertigung:=TRUE;

				IF 	gi16_maschinenstatusinfo = STATUS_BETRIEBSBEREIT THEN
					fb_state_entry.i16_next_step := FEHLER;
				END_IF
			END_IF

			(*-----------------------Weiterschaltbedingungen----------------------------*)
			IF	 i16_hubzaehler >= gst_datensatz.st_wkz.st_oeler.i16_intervall_bandoelen AND
				gst_datensatz.st_wkz.st_oeler.i16_intervall_bandoelen <>0 THEN (*bei Intervall 0 Dauerölen*)
				fb_state_entry.i16_next_step := 110;
			END_IF

		END_IF

(*=======================================================*)
	110: (* Bandölen, abhängig von WKZ-Daten *)
		IF fb_state_entry.E THEN
			i16_hubzaehler := 0;
			fb_ton_oelen.IN := TRUE;
			fb_ton_oelen.PT := DINT_TO_TIME(gst_datensatz.st_wkz.st_oeler.t_ventiloeffnungszeit);
			a_ventil := TRUE;
		END_IF

		(*-----------------------Weiterschaltbedingungen----------------------------*)
		IF fb_ton_oelen.Q THEN
			fb_ton_oelen.IN := FALSE;
			a_ventil := FALSE;
			fb_state_entry.i16_next_step := BEREIT;
		END_IF

(*=======================================================*)
	FEHLER:
		IF fb_state_entry.E THEN
			st_ctrl_out.b_fehler := TRUE;
			a_ventil := FALSE;
			fb_ton_quitt.IN := FALSE;
		END_IF

		(*-----------------------Weiterschaltbedingungen----------------------------*)
		IF st_ctrl_in.b_quitt AND NOT fb_state_entry.E THEN
			st_ctrl_out.b_fehler := FALSE;
			fb_ton_quitt.IN := TRUE;
		END_IF

		IF fb_ton_quitt.Q THEN
			fb_ton_quitt.IN := FALSE;
			fb_state_entry.i16_next_step := INIT;
		END_IF

(*=======================================================*)
	STOP:
		IF fb_state_entry.E THEN
			a_ventil := FALSE;
			fb_ton_quitt.IN := FALSE;
		END_IF

		(*-----------------------Weiterschaltbedingungen----------------------------*)
		IF st_ctrl_in.b_quitt AND NOT fb_state_entry.E THEN
			fb_ton_quitt.IN := TRUE;
		END_IF

		IF fb_ton_quitt.Q THEN
			fb_ton_quitt.IN := FALSE;
			fb_state_entry.i16_next_step := INIT;
		END_IF
END_CASE

fb_state_entry(
	i16_next_step:= , 
	i16_pos:= 2,
	s_debugtext:= ,
	E=> ,
	X=> , 
	i16_step=> ,
	i16_last_step=> );

IF st_config.b_config_fertig THEN
	(* Fehlermeldungen und Betriebsmeldungen ab dem Startindex in die globalen Meldungsarrays schreiben *)
	garr_stoermeldungen[st_config.i16_meld_startindex + 0] := sm_fuellstand_oeler;
	garr_stoermeldungen[st_config.i16_meld_startindex + 1] := sm_druckueberwachung;
	garr_stoermeldungen[st_config.i16_meld_startindex + 2] := FALSE;
	garr_stoermeldungen[st_config.i16_meld_startindex + 3] := FALSE;
	garr_stoermeldungen[st_config.i16_meld_startindex + 4] := FALSE;
	garr_stoermeldungen[st_config.i16_meld_startindex + 5] := FALSE;
	garr_stoermeldungen[st_config.i16_meld_startindex + 6] := FALSE;
	garr_stoermeldungen[st_config.i16_meld_startindex + 7] := FALSE;
	garr_stoermeldungen[st_config.i16_meld_startindex + 8] := FALSE;
	garr_stoermeldungen[st_config.i16_meld_startindex + 9] := FALSE;
	garr_stoermeldungen[st_config.i16_meld_startindex + 10] := FALSE;
	garr_stoermeldungen[st_config.i16_meld_startindex + 11] := FALSE;
	garr_stoermeldungen[st_config.i16_meld_startindex + 12] := FALSE;
	garr_stoermeldungen[st_config.i16_meld_startindex + 13] := FALSE;
	garr_stoermeldungen[st_config.i16_meld_startindex + 14] := FALSE;
	garr_stoermeldungen[st_config.i16_meld_startindex + 15] := FALSE;
	garr_stoermeldungen[st_config.i16_meld_startindex + 16] := FALSE;
	garr_stoermeldungen[st_config.i16_meld_startindex + 17] := FALSE;
	garr_stoermeldungen[st_config.i16_meld_startindex + 18] := FALSE;
	garr_stoermeldungen[st_config.i16_meld_startindex + 19] := FALSE;
	
